LIN {X 0,Y 454.422,Z 912.402,A -85,B 0,C 180,E1 7856.185,E2 7856.185} C_VEL
LIN {X 0,Y 452.901,Z 864.791,A -85,B 0,C 180,E1 7857.267,E2 7857.267} C_VEL
LIN {X 0,Y 442.42,Z 831.81,A -85,B 0,C 180,E1 7858.557,E2 7858.557} C_VEL
LIN {X 0,Y 442.033,Z 831.81,A -85,B 0,C 180,E1 7869.429,E2 7869.429} C_VEL
LIN {X 0,Y 441.898,Z 831.81,A -85,B 0,C 180,E1 7877.954,E2 7877.954} C_VEL
LIN {X 0,Y 441.923,Z 831.81,A -85,B 0,C 180,E1 7887.837,E2 7887.837} C_VEL
LIN {X 0,Y 442.333,Z 831.81,A -85,B 0,C 180,E1 7898.882,E2 7898.882} C_VEL
LIN {X 0,Y 442.705,Z 831.81,A -85,B 0,C 180,E1 7909.13,E2 7909.13} C_VEL
LIN {X 0,Y 443.019,Z 831.81,A -85,B 0,C 180,E1 7919.017,E2 7919.017} C_VEL
LIN {X 0,Y 442.99,Z 831.81,A -85,B 0,C 180,E1 7928.866,E2 7928.866} C_VEL
LIN {X 0,Y 442.447,Z 831.81,A -85,B 0,C 180,E1 7939.4,E2 7939.4} C_VEL
LIN {X 0,Y 442.141,Z 831.81,A -85,B 0,C 180,E1 7949.846,E2 7949.846} C_VEL
LIN {X 0,Y 441.891,Z 831.81,A -85,B 0,C 180,E1 7959.444,E2 7959.444} C_VEL
LIN {X 0,Y 441.878,Z 831.81,A -85,B 0,C 180,E1 7967.957,E2 7967.957} C_VEL
LIN {X 0,Y 441.956,Z 831.81,A -85,B 0,C 180,E1 7977.844,E2 7977.844} C_VEL
LIN {X 0,Y 441.962,Z 831.81,A -85,B 0,C 180,E1 7986.742,E2 7986.742} C_VEL
LIN {X 0,Y 442.386,Z 831.81,A -85,B 0,C 180,E1 7997.116,E2 7997.116} C_VEL
LIN {X 0,Y 443.102,Z 831.81,A -85,B 0,C 180,E1 8007.055,E2 8007.055} C_VEL
LIN {X 0,Y 442.319,Z 833.399,A -85,B 0,C 180,E1 8012.396,E2 8012.396} C_VEL
LIN {X 0,Y 449.483,Z 869.862,A -85,B 0,C 180,E1 8014.631,E2 8014.631} C_VEL
LIN {X 0,Y 446.798,Z 905.325,A -85,B 0,C 180,E1 8018.299,E2 8018.299} C_VEL
LIN {X 0,Y 444.934,Z 929.395,A -85,B 0,C 180,E1 8023.352,E2 8023.352} C_VEL
LIN {X 0,Y 444.173,Z 939.173,A -85,B 0,C 180,E1 8028.939,E2 8028.939} C_VEL
LIN {X 0,Y 444.716,Z 934.706,A -85,B 0,C 180,E1 8034.709,E2 8034.709} C_VEL
LIN {X 0,Y 446.355,Z 916.606,A -85,B 0,C 180,E1 8039.89,E2 8039.89} C_VEL
LIN {X 0,Y 448.943,Z 886.147,A -85,B 0,C 180,E1 8044.088,E2 8044.088} C_VEL
LIN {X 0,Y 448.622,Z 854.294,A -85,B 0,C 180,E1 8046.544,E2 8046.544} C_VEL
LIN {X 0,Y 442.206,Z 831.81,A -85,B 0,C 180,E1 8047.897,E2 8047.897} C_VEL
LIN {X 0,Y 441.835,Z 831.81,A -85,B 0,C 180,E1 8057.952,E2 8057.952} C_VEL
LIN {X 0,Y 441.941,Z 831.81,A -85,B 0,C 180,E1 8067.843,E2 8067.843} C_VEL
LIN {X 0,Y 441.947,Z 831.81,A -85,B 0,C 180,E1 8076.742,E2 8076.742} C_VEL
LIN {X 0,Y 442.404,Z 831.81,A -85,B 0,C 180,E1 8087.118,E2 8087.118} C_VEL
LIN {X 0,Y 443.089,Z 831.81,A -85,B 0,C 180,E1 8097.057,E2 8097.057} C_VEL
LIN {X 0,Y 443.038,Z 831.81,A -85,B 0,C 180,E1 8106.888,E2 8106.888} C_VEL
LIN {X 0,Y 442.488,Z 831.81,A -85,B 0,C 180,E1 8116.952,E2 8116.952} C_VEL
LIN {X 0,Y 442.171,Z 831.81,A -85,B 0,C 180,E1 8127.606,E2 8127.606} C_VEL
LIN {X 0,Y 442.046,Z 831.81,A -85,B 0,C 180,E1 8136.93,E2 8136.93} C_VEL
LIN {X 0,Y 441.891,Z 831.81,A -85,B 0,C 180,E1 8147.598,E2 8147.598} C_VEL
LIN {X 0,Y 441.964,Z 831.81,A -85,B 0,C 180,E1 8157.845,E2 8157.845} C_VEL
LIN {X 0,Y 442.599,Z 833.755,A -85,B 0,C 180,E1 8161.637,E2 8161.637} C_VEL
LIN {X 0,Y 455.096,Z 877.398,A -85,B 0,C 180,E1 8163.05,E2 8163.05} C_VEL
LIN {X 0,Y 453.053,Z 934.016,A -85,B 0,C 180,E1 8164.683,E2 8164.683} C_VEL
LIN {X 0,Y 452.974,Z 934.968,A -85,B 0,C 180,E1 8164.729,E2 8164.729} C_VEL
LIN {X 0,Y 443.094,Z 966.571,A -85,B 0,C 180,E1 8166.367,E2 8166.367} C_VEL
LIN {X 0,Y 438.906,Z 1011.784,A -85,B 0,C 180,E1 8171.012,E2 8171.012} C_VEL
LIN {X 0,Y 436.535,Z 1045.486,A -85,B 0,C 180,E1 8176.941,E2 8176.941} C_VEL
LIN {X 0,Y 435.959,Z 1065.659,A -85,B 0,C 180,E1 8183.505,E2 8183.505} C_VEL
LIN {X 0,Y 436.168,Z 1071.941,A -85,B 0,C 180,E1 8189.004,E2 8189.004} C_VEL
LIN {X 0,Y 435.757,Z 1066.82,A -85,B 0,C 180,E1 8195.934,E2 8195.934} C_VEL
LIN {X 0,Y 436.23,Z 1047.781,A -85,B 0,C 180,E1 8202.558,E2 8202.558} C_VEL
LIN {X 0,Y 438.507,Z 1016.439,A -85,B 0,C 180,E1 8208.392,E2 8208.392} C_VEL
LIN {X 0,Y 442.634,Z 972.141,A -85,B 0,C 180,E1 8213.221,E2 8213.221} C_VEL
LIN {X 0,Y 446.471,Z 920.305,A -85,B 0,C 180,E1 8216.255,E2 8216.255} C_VEL
LIN {X 0,Y 445.695,Z 867.234,A -85,B 0,C 180,E1 8217.583,E2 8217.583} C_VEL
LIN {X 0,Y 434.365,Z 831.81,A -85,B 0,C 180,E1 8218.883,E2 8218.883} C_VEL
LIN {X 0,Y 433.936,Z 831.81,A -85,B 0,C 180,E1 8228.1,E2 8228.1} C_VEL
LIN {X 0,Y 433.837,Z 831.81,A -85,B 0,C 180,E1 8238.77,E2 8238.77} C_VEL
LIN {X 0,Y 433.955,Z 831.81,A -85,B 0,C 180,E1 8249.527,E2 8249.527} C_VEL
LIN {X 0,Y 434.401,Z 831.81,A -85,B 0,C 180,E1 8260.614,E2 8260.614} C_VEL
LIN {X 0,Y 434.81,Z 831.81,A -85,B 0,C 180,E1 8270.961,E2 8270.961} C_VEL
LIN {X 0,Y 435.516,Z 831.81,A -85,B 0,C 180,E1 8280.996,E2 8280.996} C_VEL
LIN {X 0,Y 434.775,Z 831.81,A -85,B 0,C 180,E1 8291.067,E2 8291.067} C_VEL
LIN {X 0,Y 434.374,Z 831.81,A -85,B 0,C 180,E1 8301.519,E2 8301.519} C_VEL
LIN {X 0,Y 433.976,Z 831.81,A -85,B 0,C 180,E1 8311.049,E2 8311.049} C_VEL
LIN {X 0,Y 433.808,Z 831.81,A -85,B 0,C 180,E1 8321.226,E2 8321.226} C_VEL
LIN {X 0,Y 433.755,Z 831.81,A -85,B 0,C 180,E1 8331.925,E2 8331.925} C_VEL
LIN {X 0,Y 434.054,Z 831.81,A -85,B 0,C 180,E1 8341.836,E2 8341.836} C_VEL
LIN {X 0,Y 434.263,Z 831.81,A -85,B 0,C 180,E1 8352.72,E2 8352.72} C_VEL
LIN {X 0,Y 434.922,Z 831.81,A -85,B 0,C 180,E1 8362.985,E2 8362.985} C_VEL
LIN {X 0,Y 434.261,Z 831.81,A -85,B 0,C 180,E1 8371.877,E2 8371.877} C_VEL
LIN {X 0,Y 441.916,Z 870.864,A -85,B 0,C 180,E1 8374.328,E2 8374.328} C_VEL
LIN {X 0,Y 439.148,Z 905.532,A -85,B 0,C 180,E1 8377.945,E2 8377.945} C_VEL
LIN {X 0,Y 437.129,Z 929.985,A -85,B 0,C 180,E1 8383.041,E2 8383.041} C_VEL
LIN {X 0,Y 436.474,Z 938.88,A -85,B 0,C 180,E1 8387.189,E2 8387.189} C_VEL
LIN {X 0,Y 436.668,Z 938.097,A -85,B 0,C 180,E1 8393.556,E2 8393.556} C_VEL
LIN {X 0,Y 438.194,Z 922.963,A -85,B 0,C 180,E1 8399.002,E2 8399.002} C_VEL
LIN {X 0,Y 440.773,Z 895,A -85,B 0,C 180,E1 8403.574,E2 8403.574} C_VEL
LIN {X 0,Y 441.368,Z 856.806,A -85,B 0,C 180,E1 8406.828,E2 8406.828} C_VEL
LIN {X 0,Y 434.167,Z 831.81,A -85,B 0,C 180,E1 8408.449,E2 8408.449} C_VEL
LIN {X 0,Y 433.703,Z 831.81,A -85,B 0,C 180,E1 8419.66,E2 8419.66} C_VEL
LIN {X 0,Y 433.965,Z 831.81,A -85,B 0,C 180,E1 8429.533,E2 8429.533} C_VEL
LIN {X 0,Y 434.066,Z 831.81,A -85,B 0,C 180,E1 8440.603,E2 8440.603} C_VEL
LIN {X 0,Y 434.843,Z 831.81,A -85,B 0,C 180,E1 8450.966,E2 8450.966} C_VEL
LIN {X 0,Y 435.008,Z 831.81,A -85,B 0,C 180,E1 8461.001,E2 8461.001} C_VEL
LIN {X 0,Y 434.712,Z 831.81,A -85,B 0,C 180,E1 8471.072,E2 8471.072} C_VEL
LIN {X 0,Y 434.335,Z 831.81,A -85,B 0,C 180,E1 8481.526,E2 8481.526} C_VEL
LIN {X 0,Y 433.993,Z 831.81,A -85,B 0,C 180,E1 8491.054,E2 8491.054} C_VEL
LIN {X 0,Y 433.899,Z 831.81,A -85,B 0,C 180,E1 8501.241,E2 8501.241} C_VEL
LIN {X 0,Y 433.843,Z 831.81,A -85,B 0,C 180,E1 8512.257,E2 8512.257} C_VEL
LIN {X 0,Y 434.468,Z 833.594,A -85,B 0,C 180,E1 8521.146,E2 8521.146} C_VEL
LIN {X 0,Y 447.732,Z 879.445,A -85,B 0,C 180,E1 8522.688,E2 8522.688} C_VEL
LIN {X 0,Y 445.41,Z 935.367,A -85,B 0,C 180,E1 8524.403,E2 8524.403} C_VEL
LIN {X 0,Y 443.094,Z 966.571,A -85,B 0,C 180,E1 8526.367,E2 8526.367} C_VEL
LIN {X 0,Y 432.74,Z 995.144,A -85,B 0,C 180,E1 8528.771,E2 8528.771} C_VEL
LIN {X 0,Y 429.368,Z 1034.587,A -85,B 0,C 180,E1 8534.629,E2 8534.629} C_VEL
LIN {X 0,Y 427.888,Z 1059.791,A -85,B 0,C 180,E1 8541.331,E2 8541.331} C_VEL
LIN {X 0,Y 427.788,Z 1069.446,A -85,B 0,C 180,E1 8546.95,E2 8546.95} C_VEL
LIN {X 0,Y 428.088,Z 1068.529,A -85,B 0,C 180,E1 8554.066,E2 8554.066} C_VEL
LIN {X 0,Y 428.186,Z 1052.254,A -85,B 0,C 180,E1 8561.241,E2 8561.241} C_VEL
LIN {X 0,Y 430.22,Z 1021.325,A -85,B 0,C 180,E1 8567.766,E2 8567.766} C_VEL
LIN {X 0,Y 434.404,Z 978.475,A -85,B 0,C 180,E1 8572.932,E2 8572.932} C_VEL
LIN {X 0,Y 438.433,Z 927.776,A -85,B 0,C 180,E1 8576.285,E2 8576.285} C_VEL
LIN {X 0,Y 438.872,Z 870.815,A -85,B 0,C 180,E1 8577.872,E2 8577.872} C_VEL
LIN {X 0,Y 426.276,Z 831.81,A -85,B 0,C 180,E1 8579.275,E2 8579.275} C_VEL
LIN {X 0,Y 425.881,Z 831.81,A -85,B 0,C 180,E1 8589.987,E2 8589.987} C_VEL
LIN {X 0,Y 425.797,Z 831.81,A -85,B 0,C 180,E1 8600.02,E2 8600.02} C_VEL
LIN {X 0,Y 425.943,Z 831.81,A -85,B 0,C 180,E1 8611.247,E2 8611.247} C_VEL
LIN {X 0,Y 426.421,Z 831.81,A -85,B 0,C 180,E1 8622.389,E2 8622.389} C_VEL
LIN {X 0,Y 426.997,Z 831.81,A -85,B 0,C 180,E1 8632.852,E2 8632.852} C_VEL
LIN {X 0,Y 427.059,Z 831.81,A -85,B 0,C 180,E1 8643.054,E2 8643.054} C_VEL
LIN {X 0,Y 426.64,Z 831.81,A -85,B 0,C 180,E1 8653.367,E2 8653.367} C_VEL
LIN {X 0,Y 426.262,Z 831.81,A -85,B 0,C 180,E1 8664.167,E2 8664.167} C_VEL
LIN {X 0,Y 425.868,Z 831.81,A -85,B 0,C 180,E1 8673.527,E2 8673.527} C_VEL
LIN {X 0,Y 425.807,Z 831.81,A -85,B 0,C 180,E1 8684.025,E2 8684.025} C_VEL
LIN {X 0,Y 425.75,Z 831.81,A -85,B 0,C 180,E1 8693.976,E2 8693.976} C_VEL
LIN {X 0,Y 426.032,Z 831.81,A -85,B 0,C 180,E1 8703.56,E2 8703.56} C_VEL
LIN {X 0,Y 426.321,Z 831.81,A -85,B 0,C 180,E1 8714.516,E2 8714.516} C_VEL
LIN {X 0,Y 426.823,Z 831.81,A -85,B 0,C 180,E1 8724.9,E2 8724.9} C_VEL
LIN {X 0,Y 426.5,Z 833.49,A -85,B 0,C 180,E1 8731.561,E2 8731.561} C_VEL
LIN {X 0,Y 434.317,Z 872.523,A -85,B 0,C 180,E1 8734.063,E2 8734.063} C_VEL
LIN {X 0,Y 431.356,Z 907.491,A -85,B 0,C 180,E1 8737.835,E2 8737.835} C_VEL
LIN {X 0,Y 429.326,Z 930.682,A -85,B 0,C 180,E1 8742.763,E2 8742.763} C_VEL
LIN {X 0,Y 428.543,Z 940.498,A -85,B 0,C 180,E1 8747.517,E2 8747.517} C_VEL
LIN {X 0,Y 428.749,Z 939.811,A -85,B 0,C 180,E1 8753.296,E2 8753.296} C_VEL
LIN {X 0,Y 430.281,Z 925.373,A -85,B 0,C 180,E1 8758.923,E2 8758.923} C_VEL
LIN {X 0,Y 432.969,Z 898.325,A -85,B 0,C 180,E1 8763.617,E2 8763.617} C_VEL
LIN {X 0,Y 434.419,Z 860.694,A -85,B 0,C 180,E1 8767.02,E2 8767.02} C_VEL
LIN {X 0,Y 426.096,Z 831.81,A -85,B 0,C 180,E1 8768.952,E2 8768.952} C_VEL
LIN {X 0,Y 425.672,Z 831.81,A -85,B 0,C 180,E1 8780.039,E2 8780.039} C_VEL
LIN {X 0,Y 425.956,Z 831.81,A -85,B 0,C 180,E1 8791.252,E2 8791.252} C_VEL
LIN {X 0,Y 426.191,Z 831.81,A -85,B 0,C 180,E1 8802.384,E2 8802.384} C_VEL
LIN {X 0,Y 426.9,Z 831.81,A -85,B 0,C 180,E1 8812.854,E2 8812.854} C_VEL
LIN {X 0,Y 427.017,Z 831.81,A -85,B 0,C 180,E1 8821.02,E2 8821.02} C_VEL
LIN {X 0,Y 426.69,Z 831.81,A -85,B 0,C 180,E1 8831.283,E2 8831.283} C_VEL
LIN {X 0,Y 426.3,Z 831.81,A -85,B 0,C 180,E1 8841.952,E2 8841.952} C_VEL
LIN {X 0,Y 425.973,Z 831.81,A -85,B 0,C 180,E1 8853.156,E2 8853.156} C_VEL
LIN {X 0,Y 425.852,Z 831.81,A -85,B 0,C 180,E1 8864.025,E2 8864.025} C_VEL
LIN {X 0,Y 425.799,Z 831.81,A -85,B 0,C 180,E1 8873.981,E2 8873.981} C_VEL
LIN {X 0,Y 426.336,Z 833.295,A -85,B 0,C 180,E1 8880.622,E2 8880.622} C_VEL
LIN {X 0,Y 440.369,Z 881.983,A -85,B 0,C 180,E1 8882.322,E2 8882.322} C_VEL
LIN {X 0,Y 437.735,Z 937.584,A -85,B 0,C 180,E1 8884.156,E2 8884.156} C_VEL
LIN {X 0,Y 433.497,Z 987.759,A -85,B 0,C 180,E1 8887.976,E2 8887.976} C_VEL
LIN {X 0,Y 432.74,Z 995.144,A -85,B 0,C 180,E1 8888.771,E2 8888.771} C_VEL
LIN {X 0,Y 422.54,Z 1019.728,A -85,B 0,C 180,E1 8891.909,E2 8891.909} C_VEL
LIN {X 0,Y 420.47,Z 1050.799,A -85,B 0,C 180,E1 8898.551,E2 8898.551} C_VEL
LIN {X 0,Y 419.97,Z 1067.213,A -85,B 0,C 180,E1 8905.856,E2 8905.856} C_VEL
LIN {X 0,Y 419.958,Z 1069.521,A -85,B 0,C 180,E1 8911.036,E2 8911.036} C_VEL
LIN {X 0,Y 419.861,Z 1061.159,A -85,B 0,C 180,E1 8917.79,E2 8917.79} C_VEL
LIN {X 0,Y 421.193,Z 1037.3,A -85,B 0,C 180,E1 8924.875,E2 8924.875} C_VEL
LIN {X 0,Y 424.412,Z 1000.57,A -85,B 0,C 180,E1 8930.814,E2 8930.814} C_VEL
LIN {X 0,Y 428.924,Z 952.896,A -85,B 0,C 180,E1 8935.219,E2 8935.219} C_VEL
LIN {X 0,Y 432.413,Z 900.477,A -85,B 0,C 180,E1 8937.613,E2 8937.613} C_VEL
LIN {X 0,Y 430.283,Z 868.597,A -85,B 0,C 180,E1 8938.364,E2 8938.364} C_VEL
LIN {X 0,Y 418.157,Z 831.81,A -85,B 0,C 180,E1 8939.936,E2 8939.936} C_VEL
LIN {X 0,Y 417.859,Z 831.81,A -85,B 0,C 180,E1 8949.461,E2 8949.461} C_VEL
LIN {X 0,Y 417.777,Z 831.81,A -85,B 0,C 180,E1 8960.525,E2 8960.525} C_VEL
LIN {X 0,Y 417.916,Z 831.81,A -85,B 0,C 180,E1 8970.641,E2 8970.641} C_VEL
LIN {X 0,Y 418.385,Z 831.81,A -85,B 0,C 180,E1 8982.04,E2 8982.04} C_VEL
LIN {X 0,Y 418.981,Z 831.81,A -85,B 0,C 180,E1 8992.715,E2 8992.715} C_VEL
LIN {X 0,Y 419.043,Z 831.81,A -85,B 0,C 180,E1 9003.112,E2 9003.112} C_VEL
LIN {X 0,Y 418.607,Z 831.81,A -85,B 0,C 180,E1 9013.628,E2 9013.628} C_VEL
LIN {X 0,Y 418.245,Z 831.81,A -85,B 0,C 180,E1 9024.661,E2 9024.661} C_VEL
LIN {X 0,Y 417.704,Z 831.81,A -85,B 0,C 180,E1 9035.17,E2 9035.17} C_VEL
LIN {X 0,Y 417.774,Z 831.81,A -85,B 0,C 180,E1 9045.099,E2 9045.099} C_VEL
LIN {X 0,Y 417.744,Z 831.81,A -85,B 0,C 180,E1 9055.731,E2 9055.731} C_VEL
LIN {X 0,Y 417.962,Z 831.81,A -85,B 0,C 180,E1 9065.32,E2 9065.32} C_VEL
LIN {X 0,Y 418.302,Z 831.81,A -85,B 0,C 180,E1 9076.36,E2 9076.36} C_VEL
LIN {X 0,Y 419.049,Z 831.81,A -85,B 0,C 180,E1 9086.886,E2 9086.886} C_VEL
LIN {X 0,Y 418.651,Z 833.62,A -85,B 0,C 180,E1 9091.135,E2 9091.135} C_VEL
LIN {X 0,Y 426.787,Z 873.187,A -85,B 0,C 180,E1 9093.713,E2 9093.713} C_VEL
LIN {X 0,Y 423.565,Z 909.392,A -85,B 0,C 180,E1 9097.721,E2 9097.721} C_VEL
LIN {X 0,Y 421.377,Z 932.957,A -85,B 0,C 180,E1 9103.006,E2 9103.006} C_VEL
LIN {X 0,Y 420.597,Z 942.014,A -85,B 0,C 180,E1 9107.859,E2 9107.859} C_VEL
LIN {X 0,Y 421.035,Z 939.377,A -85,B 0,C 180,E1 9114.487,E2 9114.487} C_VEL
LIN {X 0,Y 423.044,Z 922.373,A -85,B 0,C 180,E1 9120.126,E2 9120.126} C_VEL
LIN {X 0,Y 426.057,Z 893.863,A -85,B 0,C 180,E1 9124.61,E2 9124.61} C_VEL
LIN {X 0,Y 426.409,Z 859.686,A -85,B 0,C 180,E1 9127.602,E2 9127.602} C_VEL
LIN {X 0,Y 418.049,Z 831.81,A -85,B 0,C 180,E1 9129.439,E2 9129.439} C_VEL
LIN {X 0,Y 417.647,Z 831.81,A -85,B 0,C 180,E1 9140.515,E2 9140.515} C_VEL
LIN {X 0,Y 417.926,Z 831.81,A -85,B 0,C 180,E1 9150.647,E2 9150.647} C_VEL
LIN {X 0,Y 418.138,Z 831.81,A -85,B 0,C 180,E1 9162.033,E2 9162.033} C_VEL
LIN {X 0,Y 418.878,Z 831.81,A -85,B 0,C 180,E1 9172.717,E2 9172.717} C_VEL
LIN {X 0,Y 419.011,Z 831.81,A -85,B 0,C 180,E1 9181.04,E2 9181.04} C_VEL
LIN {X 0,Y 418.687,Z 831.81,A -85,B 0,C 180,E1 9191.502,E2 9191.502} C_VEL
LIN {X 0,Y 418.234,Z 831.81,A -85,B 0,C 180,E1 9202.398,E2 9202.398} C_VEL
LIN {X 0,Y 417.923,Z 831.81,A -85,B 0,C 180,E1 9211.775,E2 9211.775} C_VEL
LIN {X 0,Y 417.855,Z 831.81,A -85,B 0,C 180,E1 9222.218,E2 9222.218} C_VEL
LIN {X 0,Y 417.783,Z 831.81,A -85,B 0,C 180,E1 9233.178,E2 9233.178} C_VEL
LIN {X 0,Y 418.293,Z 833.427,A -85,B 0,C 180,E1 9240.09,E2 9240.09} C_VEL
LIN {X 0,Y 433.058,Z 882.531,A -85,B 0,C 180,E1 9241.906,E2 9241.906} C_VEL
LIN {X 0,Y 430.285,Z 936.811,A -85,B 0,C 180,E1 9243.747,E2 9243.747} C_VEL
LIN {X 0,Y 425.892,Z 986,A -85,B 0,C 180,E1 9247.534,E2 9247.534} C_VEL
LIN {X 0,Y 422.54,Z 1019.728,A -85,B 0,C 180,E1 9251.909,E2 9251.909} C_VEL
LIN {X 0,Y 412.802,Z 1039.684,A -85,B 0,C 180,E1 9255.728,E2 9255.728} C_VEL
LIN {X 0,Y 412.014,Z 1060.915,A -85,B 0,C 180,E1 9262.594,E2 9262.594} C_VEL
LIN {X 0,Y 412.387,Z 1068.355,A -85,B 0,C 180,E1 9268.946,E2 9268.946} C_VEL
LIN {X 0,Y 411.912,Z 1063.046,A -85,B 0,C 180,E1 9276.351,E2 9276.351} C_VEL
LIN {X 0,Y 412.463,Z 1044.474,A -85,B 0,C 180,E1 9283.123,E2 9283.123} C_VEL
LIN {X 0,Y 414.97,Z 1013.498,A -85,B 0,C 180,E1 9289.216,E2 9289.216} C_VEL
LIN {X 0,Y 419.687,Z 969.196,A -85,B 0,C 180,E1 9294.287,E2 9294.287} C_VEL
LIN {X 0,Y 424.093,Z 917.458,A -85,B 0,C 180,E1 9297.432,E2 9297.432} C_VEL
LIN {X 0,Y 423.379,Z 871.81,A -85,B 0,C 180,E1 9298.683,E2 9298.683} C_VEL
LIN {X 0,Y 410.125,Z 831.81,A -85,B 0,C 180,E1 9300.234,E2 9300.234} C_VEL
LIN {X 0,Y 409.773,Z 831.81,A -85,B 0,C 180,E1 9310.6,E2 9310.6} C_VEL
LIN {X 0,Y 409.709,Z 831.81,A -85,B 0,C 180,E1 9319.589,E2 9319.589} C_VEL
LIN {X 0,Y 409.896,Z 831.81,A -85,B 0,C 180,E1 9330.463,E2 9330.463} C_VEL
LIN {X 0,Y 410.325,Z 831.81,A -85,B 0,C 180,E1 9341.674,E2 9341.674} C_VEL
LIN {X 0,Y 410.944,Z 831.81,A -85,B 0,C 180,E1 9352.571,E2 9352.571} C_VEL
LIN {X 0,Y 411.04,Z 831.81,A -85,B 0,C 180,E1 9363.173,E2 9363.173} C_VEL
LIN {X 0,Y 410.57,Z 831.81,A -85,B 0,C 180,E1 9373.9,E2 9373.9} C_VEL
LIN {X 0,Y 410.153,Z 831.81,A -85,B 0,C 180,E1 9385.181,E2 9385.181} C_VEL
LIN {X 0,Y 409.708,Z 831.81,A -85,B 0,C 180,E1 9395.037,E2 9395.037} C_VEL
LIN {X 0,Y 409.67,Z 831.81,A -85,B 0,C 180,E1 9406.248,E2 9406.248} C_VEL
LIN {X 0,Y 409.747,Z 831.81,A -85,B 0,C 180,E1 9417.518,E2 9417.518} C_VEL
LIN {X 0,Y 409.854,Z 831.81,A -85,B 0,C 180,E1 9427.121,E2 9427.121} C_VEL
LIN {X 0,Y 410.464,Z 831.81,A -85,B 0,C 180,E1 9438.454,E2 9438.454} C_VEL
LIN {X 0,Y 411.311,Z 831.81,A -85,B 0,C 180,E1 9448.943,E2 9448.943} C_VEL
LIN {X 0,Y 410.796,Z 833.812,A -85,B 0,C 180,E1 9450.694,E2 9450.694} C_VEL
LIN {X 0,Y 419.233,Z 874.42,A -85,B 0,C 180,E1 9453.402,E2 9453.402} C_VEL
LIN {X 0,Y 415.938,Z 909.617,A -85,B 0,C 180,E1 9457.336,E2 9457.336} C_VEL
LIN {X 0,Y 413.628,Z 933.1,A -85,B 0,C 180,E1 9462.526,E2 9462.526} C_VEL
LIN {X 0,Y 412.652,Z 943.528,A -85,B 0,C 180,E1 9468.215,E2 9468.215} C_VEL
LIN {X 0,Y 413.255,Z 939.955,A -85,B 0,C 180,E1 9474.979,E2 9474.979} C_VEL
LIN {X 0,Y 415.541,Z 921.312,A -85,B 0,C 180,E1 9480.882,E2 9480.882} C_VEL
LIN {X 0,Y 419.021,Z 890.846,A -85,B 0,C 180,E1 9485.425,E2 9485.425} C_VEL
LIN {X 0,Y 418.779,Z 860.336,A -85,B 0,C 180,E1 9488.073,E2 9488.073} C_VEL
LIN {X 0,Y 409.908,Z 831.81,A -85,B 0,C 180,E1 9490.167,E2 9490.167} C_VEL
LIN {X 0,Y 409.605,Z 831.81,A -85,B 0,C 180,E1 9499.582,E2 9499.582} C_VEL
LIN {X 0,Y 409.917,Z 831.81,A -85,B 0,C 180,E1 9510.456,E2 9510.456} C_VEL
LIN {X 0,Y 410.06,Z 831.81,A -85,B 0,C 180,E1 9521.666,E2 9521.666} C_VEL
LIN {X 0,Y 410.849,Z 831.81,A -85,B 0,C 180,E1 9532.574,E2 9532.574} C_VEL
LIN {X 0,Y 411.02,Z 831.81,A -85,B 0,C 180,E1 9541.06,E2 9541.06} C_VEL
LIN {X 0,Y 410.679,Z 831.81,A -85,B 0,C 180,E1 9551.729,E2 9551.729} C_VEL
LIN {X 0,Y 410.169,Z 831.81,A -85,B 0,C 180,E1 9562.864,E2 9562.864} C_VEL
LIN {X 0,Y 409.818,Z 831.81,A -85,B 0,C 180,E1 9573.575,E2 9573.575} C_VEL
LIN {X 0,Y 409.714,Z 831.81,A -85,B 0,C 180,E1 9583.759,E2 9583.759} C_VEL
LIN {X 0,Y 409.737,Z 831.81,A -85,B 0,C 180,E1 9594.966,E2 9594.966} C_VEL
LIN {X 0,Y 410.286,Z 833.663,A -85,B 0,C 180,E1 9599.527,E2 9599.527} C_VEL
LIN {X 0,Y 425.783,Z 883.698,A -85,B 0,C 180,E1 9601.48,E2 9601.48} C_VEL
LIN {X 0,Y 422.731,Z 937.734,A -85,B 0,C 180,E1 9603.41,E2 9603.41} C_VEL
LIN {X 0,Y 417.973,Z 987.695,A -85,B 0,C 180,E1 9607.45,E2 9607.45} C_VEL
LIN {X 0,Y 414.091,Z 1028.005,A -85,B 0,C 180,E1 9613.26,E2 9613.26} C_VEL
LIN {X 0,Y 412.802,Z 1039.684,A -85,B 0,C 180,E1 9615.728,E2 9615.728} C_VEL
LIN {X 0,Y 404.265,Z 1054.28,A -85,B 0,C 180,E1 9620.126,E2 9620.126} C_VEL
LIN {X 0,Y 404.059,Z 1065.854,A -85,B 0,C 180,E1 9626.771,E2 9626.771} C_VEL
LIN {X 0,Y 404.291,Z 1064.897,A -85,B 0,C 180,E1 9634.306,E2 9634.306} C_VEL
LIN {X 0,Y 404.267,Z 1050.07,A -85,B 0,C 180,E1 9641.366,E2 9641.366} C_VEL
LIN {X 0,Y 406.332,Z 1021.45,A -85,B 0,C 180,E1 9648.022,E2 9648.022} C_VEL
LIN {X 0,Y 410.897,Z 980.22,A -85,B 0,C 180,E1 9653.537,E2 9653.537} C_VEL
LIN {X 0,Y 415.595,Z 930.179,A -85,B 0,C 180,E1 9657.231,E2 9657.231} C_VEL
LIN {X 0,Y 416.669,Z 875.936,A -85,B 0,C 180,E1 9658.978,E2 9658.978} C_VEL
LIN {X 0,Y 402.095,Z 831.81,A -85,B 0,C 180,E1 9660.631,E2 9660.631} C_VEL
LIN {X 0,Y 401.674,Z 831.81,A -85,B 0,C 180,E1 9671.389,E2 9671.389} C_VEL
LIN {X 0,Y 401.642,Z 831.81,A -85,B 0,C 180,E1 9681.428,E2 9681.428} C_VEL
LIN {X 0,Y 401.909,Z 831.81,A -85,B 0,C 180,E1 9692.539,E2 9692.539} C_VEL
LIN {X 0,Y 402.484,Z 831.81,A -85,B 0,C 180,E1 9704.043,E2 9704.043} C_VEL
LIN {X 0,Y 402.993,Z 831.81,A -85,B 0,C 180,E1 9714.596,E2 9714.596} C_VEL
LIN {X 0,Y 402.951,Z 831.81,A -85,B 0,C 180,E1 9723.613,E2 9723.613} C_VEL
LIN {X 0,Y 402.535,Z 831.81,A -85,B 0,C 180,E1 9734.183,E2 9734.183} C_VEL
LIN {X 0,Y 402.066,Z 831.81,A -85,B 0,C 180,E1 9745.724,E2 9745.724} C_VEL
LIN {X 0,Y 401.646,Z 831.81,A -85,B 0,C 180,E1 9755.848,E2 9755.848} C_VEL
LIN {X 0,Y 401.608,Z 831.81,A -85,B 0,C 180,E1 9765.649,E2 9765.649} C_VEL
LIN {X 0,Y 401.711,Z 831.81,A -85,B 0,C 180,E1 9776.786,E2 9776.786} C_VEL
LIN {X 0,Y 401.837,Z 831.81,A -85,B 0,C 180,E1 9787.708,E2 9787.708} C_VEL
LIN {X 0,Y 402.392,Z 831.81,A -85,B 0,C 180,E1 9798.028,E2 9798.028} C_VEL
LIN {X 0,Y 403.301,Z 831.81,A -85,B 0,C 180,E1 9808.922,E2 9808.922} C_VEL
LIN {X 0,Y 403.002,Z 833.939,A -85,B 0,C 180,E1 9810.236,E2 9810.236} C_VEL
LIN {X 0,Y 411.716,Z 875.082,A -85,B 0,C 180,E1 9813.038,E2 9813.038} C_VEL
LIN {X 0,Y 408.14,Z 911.447,A -85,B 0,C 180,E1 9817.209,E2 9817.209} C_VEL
LIN {X 0,Y 405.721,Z 935.024,A -85,B 0,C 180,E1 9822.664,E2 9822.664} C_VEL
LIN {X 0,Y 404.734,Z 944.938,A -85,B 0,C 180,E1 9828.584,E2 9828.584} C_VEL
LIN {X 0,Y 405.447,Z 940.499,A -85,B 0,C 180,E1 9835.494,E2 9835.494} C_VEL
LIN {X 0,Y 407.953,Z 921.631,A -85,B 0,C 180,E1 9841.344,E2 9841.344} C_VEL
LIN {X 0,Y 411.719,Z 890.66,A -85,B 0,C 180,E1 9845.945,E2 9845.945} C_VEL
LIN {X 0,Y 411.583,Z 862.876,A -85,B 0,C 180,E1 9848.416,E2 9848.416} C_VEL
LIN {X 0,Y 401.812,Z 831.81,A -85,B 0,C 180,E1 9850.931,E2 9850.931} C_VEL
LIN {X 0,Y 401.499,Z 831.81,A -85,B 0,C 180,E1 9861.417,E2 9861.417} C_VEL
LIN {X 0,Y 401.911,Z 831.81,A -85,B 0,C 180,E1 9872.537,E2 9872.537} C_VEL
LIN {X 0,Y 402.229,Z 831.81,A -85,B 0,C 180,E1 9884.167,E2 9884.167} C_VEL
LIN {X 0,Y 402.806,Z 831.81,A -85,B 0,C 180,E1 9894.597,E2 9894.597} C_VEL
LIN {X 0,Y 402.879,Z 831.81,A -85,B 0,C 180,E1 9903.46,E2 9903.46} C_VEL
LIN {X 0,Y 402.543,Z 831.81,A -85,B 0,C 180,E1 9914.187,E2 9914.187} C_VEL
LIN {X 0,Y 402.023,Z 831.81,A -85,B 0,C 180,E1 9925.732,E2 9925.732} C_VEL
LIN {X 0,Y 401.798,Z 831.81,A -85,B 0,C 180,E1 9935.837,E2 9935.837} C_VEL
LIN {X 0,Y 401.638,Z 831.81,A -85,B 0,C 180,E1 9945.654,E2 9945.654} C_VEL
LIN {X 0,Y 401.736,Z 831.81,A -85,B 0,C 180,E1 9956.789,E2 9956.789} C_VEL
LIN {X 0,Y 402.193,Z 833.57,A -85,B 0,C 180,E1 9958.92,E2 9958.92} C_VEL
LIN {X 0,Y 418.532,Z 883.85,A -85,B 0,C 180,E1 9961.021,E2 9961.021} C_VEL
LIN {X 0,Y 415.326,Z 937.504,A -85,B 0,C 180,E1 9962.994,E2 9962.994} C_VEL
LIN {X 0,Y 410.358,Z 986.281,A -85,B 0,C 180,E1 9967.008,E2 9967.008} C_VEL
LIN {X 0,Y 406.217,Z 1026.846,A -85,B 0,C 180,E1 9972.955,E2 9972.955} C_VEL
LIN {X 0,Y 404.265,Z 1054.28,A -85,B 0,C 180,E1 9980.126,E2 9980.126} C_VEL
LIN {X 0,Y 396.284,Z 1062.81,A -85,B 0,C 180,E1 9984.942,E2 9984.942} C_VEL
LIN {X 0,Y 396.225,Z 1065.94,A -85,B 0,C 180,E1 9991.098,E2 9991.098} C_VEL
LIN {X 0,Y 396.115,Z 1057.386,A -85,B 0,C 180,E1 9998.26,E2 9998.26} C_VEL
LIN {X 0,Y 397.702,Z 1033.036,A -85,B 0,C 180,E1 10005.776,E2 10005.776} C_VEL
LIN {X 0,Y 401.455,Z 995.539,A -85,B 0,C 180,E1 10012.04,E2 10012.04} C_VEL
LIN {X 0,Y 406.55,Z 947.581,A -85,B 0,C 180,E1 10016.557,E2 10016.557} C_VEL
LIN {X 0,Y 410.233,Z 895.116,A -85,B 0,C 180,E1 10018.932,E2 10018.932} C_VEL
LIN {X 0,Y 407.173,Z 870.658,A -85,B 0,C 180,E1 10019.612,E2 10019.612} C_VEL
LIN {X 0,Y 393.963,Z 831.81,A -85,B 0,C 180,E1 10021.334,E2 10021.334} C_VEL
LIN {X 0,Y 393.659,Z 831.81,A -85,B 0,C 180,E1 10032.425,E2 10032.425} C_VEL
LIN {X 0,Y 393.567,Z 831.81,A -85,B 0,C 180,E1 10043.292,E2 10043.292} C_VEL
LIN {X 0,Y 393.871,Z 831.81,A -85,B 0,C 180,E1 10053.695,E2 10053.695} C_VEL
LIN {X 0,Y 394.539,Z 831.81,A -85,B 0,C 180,E1 10065.519,E2 10065.519} C_VEL
LIN {X 0,Y 394.919,Z 831.81,A -85,B 0,C 180,E1 10076.693,E2 10076.693} C_VEL
LIN {X 0,Y 394.814,Z 831.81,A -85,B 0,C 180,E1 10085.512,E2 10085.512} C_VEL
LIN {X 0,Y 394.46,Z 831.81,A -85,B 0,C 180,E1 10096.769,E2 10096.769} C_VEL
LIN {X 0,Y 394.028,Z 831.81,A -85,B 0,C 180,E1 10106.289,E2 10106.289} C_VEL
LIN {X 0,Y 393.522,Z 831.81,A -85,B 0,C 180,E1 10117.763,E2 10117.763} C_VEL
LIN {X 0,Y 393.554,Z 831.81,A -85,B 0,C 180,E1 10128.757,E2 10128.757} C_VEL
LIN {X 0,Y 393.721,Z 831.81,A -85,B 0,C 180,E1 10140.14,E2 10140.14} C_VEL
LIN {X 0,Y 393.939,Z 831.81,A -85,B 0,C 180,E1 10150.886,E2 10150.886} C_VEL
LIN {X 0,Y 394.783,Z 831.81,A -85,B 0,C 180,E1 10162.268,E2 10162.268} C_VEL
LIN {X 0,Y 395.022,Z 833.052,A -85,B 0,C 180,E1 10169.724,E2 10169.724} C_VEL
LIN {X 0,Y 404.224,Z 875.741,A -85,B 0,C 180,E1 10172.661,E2 10172.661} C_VEL
LIN {X 0,Y 400.58,Z 911.608,A -85,B 0,C 180,E1 10176.799,E2 10176.799} C_VEL
LIN {X 0,Y 398.016,Z 934.968,A -85,B 0,C 180,E1 10182.104,E2 10182.104} C_VEL
LIN {X 0,Y 397.081,Z 944.396,A -85,B 0,C 180,E1 10186.656,E2 10186.656} C_VEL
LIN {X 0,Y 396.863,Z 946.437,A -85,B 0,C 180,E1 10191.3,E2 10191.3} C_VEL
LIN {X 0,Y 398.222,Z 936.677,A -85,B 0,C 180,E1 10197.852,E2 10197.852} C_VEL
LIN {X 0,Y 401.482,Z 913.185,A -85,B 0,C 180,E1 10203.477,E2 10203.477} C_VEL
LIN {X 0,Y 405.58,Z 877.859,A -85,B 0,C 180,E1 10207.687,E2 10207.687} C_VEL
LIN {X 0,Y 397.574,Z 842.646,A -85,B 0,C 180,E1 10210.568,E2 10210.568} C_VEL
LIN {X 0,Y 393.762,Z 831.81,A -85,B 0,C 180,E1 10211.277,E2 10211.277} C_VEL
LIN {X 0,Y 393.432,Z 831.81,A -85,B 0,C 180,E1 10222.252,E2 10222.252} C_VEL
LIN {X 0,Y 393.852,Z 831.81,A -85,B 0,C 180,E1 10233.699,E2 10233.699} C_VEL
LIN {X 0,Y 394.23,Z 831.81,A -85,B 0,C 180,E1 10245.511,E2 10245.511} C_VEL
LIN {X 0,Y 395.024,Z 831.81,A -85,B 0,C 180,E1 10256.699,E2 10256.699} C_VEL
LIN {X 0,Y 394.883,Z 831.81,A -85,B 0,C 180,E1 10267.733,E2 10267.733} C_VEL
LIN {X 0,Y 394.248,Z 831.81,A -85,B 0,C 180,E1 10279.101,E2 10279.101} C_VEL
LIN {X 0,Y 393.802,Z 831.81,A -85,B 0,C 180,E1 10289.883,E2 10289.883} C_VEL
LIN {X 0,Y 393.652,Z 831.81,A -85,B 0,C 180,E1 10301.26,E2 10301.26} C_VEL
LIN {X 0,Y 393.558,Z 831.81,A -85,B 0,C 180,E1 10312.237,E2 10312.237} C_VEL
LIN {X 0,Y 394.058,Z 833.428,A -85,B 0,C 180,E1 10318.279,E2 10318.279} C_VEL
LIN {X 0,Y 411.329,Z 883.93,A -85,B 0,C 180,E1 10320.544,E2 10320.544} C_VEL
LIN {X 0,Y 407.89,Z 937.583,A -85,B 0,C 180,E1 10322.58,E2 10322.58} C_VEL
LIN {X 0,Y 402.647,Z 986.127,A -85,B 0,C 180,E1 10326.689,E2 10326.689} C_VEL
LIN {X 0,Y 398.318,Z 1025.921,A -85,B 0,C 180,E1 10332.684,E2 10332.684} C_VEL
LIN {X 0,Y 396.316,Z 1053.59,A -85,B 0,C 180,E1 10340.129,E2 10340.129} C_VEL
LIN {X 0,Y 396.284,Z 1062.81,A -85,B 0,C 180,E1 10344.942,E2 10344.942} C_VEL
LIN {X 0,Y 388.381,Z 1064.754,A -85,B 0,C 180,E1 10349.988,E2 10349.988} C_VEL
LIN {X 0,Y 388.098,Z 1058.297,A -85,B 0,C 180,E1 10357.301,E2 10357.301} C_VEL
LIN {X 0,Y 389.063,Z 1037.513,A -85,B 0,C 180,E1 10364.687,E2 10364.687} C_VEL
LIN {X 0,Y 392.74,Z 1001.917,A -85,B 0,C 180,E1 10371.387,E2 10371.387} C_VEL
LIN {X 0,Y 397.95,Z 956.706,A -85,B 0,C 180,E1 10376.232,E2 10376.232} C_VEL
LIN {X 0,Y 402.455,Z 904.005,A -85,B 0,C 180,E1 10379.086,E2 10379.086} C_VEL
LIN {X 0,Y 400.759,Z 875.43,A -85,B 0,C 180,E1 10379.907,E2 10379.907} C_VEL
LIN {X 0,Y 385.881,Z 831.81,A -85,B 0,C 180,E1 10381.739,E2 10381.739} C_VEL
LIN {X 0,Y 385.627,Z 831.81,A -85,B 0,C 180,E1 10393.525,E2 10393.525} C_VEL
LIN {X 0,Y 385.547,Z 831.81,A -85,B 0,C 180,E1 10405.194,E2 10405.194} C_VEL
LIN {X 0,Y 385.897,Z 831.81,A -85,B 0,C 180,E1 10415.608,E2 10415.608} C_VEL
LIN {X 0,Y 386.476,Z 831.81,A -85,B 0,C 180,E1 10425.21,E2 10425.21} C_VEL
LIN {X 0,Y 386.932,Z 831.81,A -85,B 0,C 180,E1 10436.625,E2 10436.625} C_VEL
LIN {X 0,Y 386.833,Z 831.81,A -85,B 0,C 180,E1 10445.626,E2 10445.626} C_VEL
LIN {X 0,Y 386.399,Z 831.81,A -85,B 0,C 180,E1 10457.13,E2 10457.13} C_VEL
LIN {X 0,Y 385.872,Z 831.81,A -85,B 0,C 180,E1 10467.764,E2 10467.764} C_VEL
LIN {X 0,Y 385.535,Z 831.81,A -85,B 0,C 180,E1 10479.864,E2 10479.864} C_VEL
LIN {X 0,Y 385.507,Z 831.81,A -85,B 0,C 180,E1 10490.141,E2 10490.141} C_VEL
LIN {X 0,Y 385.726,Z 831.81,A -85,B 0,C 180,E1 10500.542,E2 10500.542} C_VEL
LIN {X 0,Y 385.894,Z 831.81,A -85,B 0,C 180,E1 10510.472,E2 10510.472} C_VEL
LIN {X 0,Y 386.747,Z 831.81,A -85,B 0,C 180,E1 10522.106,E2 10522.106} C_VEL
LIN {X 0,Y 387.325,Z 833.718,A -85,B 0,C 180,E1 10529.262,E2 10529.262} C_VEL
LIN {X 0,Y 396.767,Z 875.85,A -85,B 0,C 180,E1 10532.225,E2 10532.225} C_VEL
LIN {X 0,Y 393.005,Z 911.728,A -85,B 0,C 180,E1 10536.373,E2 10536.373} C_VEL
LIN {X 0,Y 390.236,Z 935.579,A -85,B 0,C 180,E1 10541.78,E2 10541.78} C_VEL
LIN {X 0,Y 389.084,Z 946.177,A -85,B 0,C 180,E1 10547.14,E2 10547.14} C_VEL
LIN {X 0,Y 389.451,Z 945.448,A -85,B 0,C 180,E1 10554.151,E2 10554.151} C_VEL
LIN {X 0,Y 391.971,Z 929.851,A -85,B 0,C 180,E1 10560.542,E2 10560.542} C_VEL
LIN {X 0,Y 395.986,Z 901.243,A -85,B 0,C 180,E1 10565.772,E2 10565.772} C_VEL
LIN {X 0,Y 397.245,Z 867.797,A -85,B 0,C 180,E1 10569.154,E2 10569.154} C_VEL
LIN {X 0,Y 385.658,Z 831.81,A -85,B 0,C 180,E1 10572.208,E2 10572.208} C_VEL
LIN {X 0,Y 385.433,Z 831.81,A -85,B 0,C 180,E1 10583.816,E2 10583.816} C_VEL
LIN {X 0,Y 385.761,Z 831.81,A -85,B 0,C 180,E1 10593.103,E2 10593.103} C_VEL
LIN {X 0,Y 386.177,Z 831.81,A -85,B 0,C 180,E1 10605.203,E2 10605.203} C_VEL
LIN {X 0,Y 387.022,Z 831.81,A -85,B 0,C 180,E1 10616.63,E2 10616.63} C_VEL
LIN {X 0,Y 386.846,Z 831.81,A -85,B 0,C 180,E1 10627.894,E2 10627.894} C_VEL
LIN {X 0,Y 386.219,Z 831.81,A -85,B 0,C 180,E1 10639.514,E2 10639.514} C_VEL
LIN {X 0,Y 385.84,Z 831.81,A -85,B 0,C 180,E1 10649.453,E2 10649.453} C_VEL
LIN {X 0,Y 385.612,Z 831.81,A -85,B 0,C 180,E1 10660.498,E2 10660.498} C_VEL
LIN {X 0,Y 385.565,Z 831.81,A -85,B 0,C 180,E1 10670.137,E2 10670.137} C_VEL
LIN {X 0,Y 385.978,Z 833.558,A -85,B 0,C 180,E1 10677.601,E2 10677.601} C_VEL
LIN {X 0,Y 404.188,Z 885.852,A -85,B 0,C 180,E1 10680.079,E2 10680.079} C_VEL
LIN {X 0,Y 400.342,Z 939.314,A -85,B 0,C 180,E1 10682.249,E2 10682.249} C_VEL
LIN {X 0,Y 394.789,Z 987.262,A -85,B 0,C 180,E1 10686.508,E2 10686.508} C_VEL
LIN {X 0,Y 390.34,Z 1026.164,A -85,B 0,C 180,E1 10692.627,E2 10692.627} C_VEL
LIN {X 0,Y 388.394,Z 1052.241,A -85,B 0,C 180,E1 10699.874,E2 10699.874} C_VEL
LIN {X 0,Y 388.242,Z 1063.479,A -85,B 0,C 180,E1 10706.639,E2 10706.639} C_VEL
LIN {X 0,Y 388.381,Z 1064.754,A -85,B 0,C 180,E1 10709.988,E2 10709.988} C_VEL
LIN {X 0,Y 380.356,Z 1060.541,A -85,B 0,C 180,E1 10715.123,E2 10715.123} C_VEL
LIN {X 0,Y 380.445,Z 1044.196,A -85,B 0,C 180,E1 10722.673,E2 10722.673} C_VEL
LIN {X 0,Y 383.177,Z 1013.855,A -85,B 0,C 180,E1 10729.672,E2 10729.672} C_VEL
LIN {X 0,Y 388.595,Z 971.141,A -85,B 0,C 180,E1 10735.286,E2 10735.286} C_VEL
LIN {X 0,Y 393.846,Z 920.558,A -85,B 0,C 180,E1 10738.849,E2 10738.849} C_VEL
LIN {X 0,Y 393.753,Z 878.281,A -85,B 0,C 180,E1 10740.273,E2 10740.273} C_VEL
LIN {X 0,Y 377.823,Z 831.81,A -85,B 0,C 180,E1 10742.304,E2 10742.304} C_VEL
LIN {X 0,Y 377.512,Z 831.81,A -85,B 0,C 180,E1 10751.948,E2 10751.948} C_VEL
LIN {X 0,Y 377.498,Z 831.81,A -85,B 0,C 180,E1 10761.62,E2 10761.62} C_VEL
LIN {X 0,Y 377.744,Z 831.81,A -85,B 0,C 180,E1 10772.479,E2 10772.479} C_VEL
LIN {X 0,Y 378.242,Z 831.81,A -85,B 0,C 180,E1 10782.484,E2 10782.484} C_VEL
LIN {X 0,Y 378.943,Z 831.81,A -85,B 0,C 180,E1 10794.251,E2 10794.251} C_VEL
LIN {X 0,Y 379.009,Z 831.81,A -85,B 0,C 180,E1 10803.441,E2 10803.441} C_VEL
LIN {X 0,Y 378.464,Z 831.81,A -85,B 0,C 180,E1 10815.106,E2 10815.106} C_VEL
LIN {X 0,Y 377.939,Z 831.81,A -85,B 0,C 180,E1 10825.385,E2 10825.385} C_VEL
LIN {X 0,Y 377.489,Z 831.81,A -85,B 0,C 180,E1 10835.655,E2 10835.655} C_VEL
LIN {X 0,Y 377.418,Z 831.81,A -85,B 0,C 180,E1 10845.279,E2 10845.279} C_VEL
LIN {X 0,Y 377.552,Z 831.81,A -85,B 0,C 180,E1 10857.137,E2 10857.137} C_VEL
LIN {X 0,Y 377.773,Z 831.81,A -85,B 0,C 180,E1 10867.565,E2 10867.565} C_VEL
LIN {X 0,Y 378.516,Z 831.81,A -85,B 0,C 180,E1 10879.606,E2 10879.606} C_VEL
LIN {X 0,Y 379.407,Z 833.177,A -85,B 0,C 180,E1 10888.725,E2 10888.725} C_VEL
LIN {X 0,Y 389.262,Z 876.439,A -85,B 0,C 180,E1 10891.821,E2 10891.821} C_VEL
LIN {X 0,Y 385.443,Z 911.772,A -85,B 0,C 180,E1 10895.932,E2 10895.932} C_VEL
LIN {X 0,Y 382.443,Z 936.164,A -85,B 0,C 180,E1 10901.443,E2 10901.443} C_VEL
LIN {X 0,Y 381.15,Z 947.623,A -85,B 0,C 180,E1 10907.374,E2 10907.374} C_VEL
LIN {X 0,Y 381.365,Z 947.891,A -85,B 0,C 180,E1 10913.112,E2 10913.112} C_VEL
LIN {X 0,Y 383.555,Z 935.205,A -85,B 0,C 180,E1 10919.641,E2 10919.641} C_VEL
LIN {X 0,Y 387.593,Z 909.112,A -85,B 0,C 180,E1 10925.232,E2 10925.232} C_VEL
LIN {X 0,Y 390.614,Z 872.825,A -85,B 0,C 180,E1 10929.287,E2 10929.287} C_VEL
LIN {X 0,Y 377.602,Z 831.81,A -85,B 0,C 180,E1 10932.769,E2 10932.769} C_VEL
LIN {X 0,Y 377.427,Z 831.81,A -85,B 0,C 180,E1 10944.338,E2 10944.338} C_VEL
LIN {X 0,Y 377.727,Z 831.81,A -85,B 0,C 180,E1 10955.05,E2 10955.05} C_VEL
LIN {X 0,Y 378.156,Z 831.81,A -85,B 0,C 180,E1 10964.881,E2 10964.881} C_VEL
LIN {X 0,Y 379.001,Z 831.81,A -85,B 0,C 180,E1 10976.559,E2 10976.559} C_VEL
LIN {X 0,Y 378.81,Z 831.81,A -85,B 0,C 180,E1 10988.063,E2 10988.063} C_VEL
LIN {X 0,Y 378.148,Z 831.81,A -85,B 0,C 180,E1 10999.948,E2 10999.948} C_VEL
LIN {X 0,Y 377.723,Z 831.81,A -85,B 0,C 180,E1 11010.257,E2 11010.257} C_VEL
LIN {X 0,Y 377.505,Z 831.81,A -85,B 0,C 180,E1 11021.954,E2 11021.954} C_VEL
LIN {X 0,Y 377.497,Z 831.81,A -85,B 0,C 180,E1 11031.627,E2 11031.627} C_VEL
LIN {X 0,Y 377.983,Z 833.733,A -85,B 0,C 180,E1 11036.895,E2 11036.895} C_VEL
LIN {X 0,Y 397.06,Z 886.732,A -85,B 0,C 180,E1 11039.573,E2 11039.573} C_VEL
LIN {X 0,Y 392.912,Z 940.146,A -85,B 0,C 180,E1 11041.841,E2 11041.841} C_VEL
LIN {X 0,Y 387.008,Z 987.898,A -85,B 0,C 180,E1 11046.258,E2 11046.258} C_VEL
LIN {X 0,Y 382.321,Z 1026.938,A -85,B 0,C 180,E1 11052.681,E2 11052.681} C_VEL
LIN {X 0,Y 380.382,Z 1052.477,A -85,B 0,C 180,E1 11060.239,E2 11060.239} C_VEL
LIN {X 0,Y 380.32,Z 1062.288,A -85,B 0,C 180,E1 11066.569,E2 11066.569} C_VEL
LIN {X 0,Y 380.426,Z 1062.278,A -85,B 0,C 180,E1 11073.431,E2 11073.431} C_VEL
LIN {X 0,Y 380.356,Z 1060.541,A -85,B 0,C 180,E1 11075.123,E2 11075.123} C_VEL
LIN {X 0,Y 372.51,Z 1050.437,A -85,B 0,C 180,E1 11080.18,E2 11080.18} C_VEL
LIN {X 0,Y 374.252,Z 1024.481,A -85,B 0,C 180,E1 11087.705,E2 11087.705} C_VEL
LIN {X 0,Y 379.192,Z 985.015,A -85,B 0,C 180,E1 11094.061,E2 11094.061} C_VEL
LIN {X 0,Y 384.866,Z 936.21,A -85,B 0,C 180,E1 11098.401,E2 11098.401} C_VEL
LIN {X 0,Y 387.519,Z 883.62,A -85,B 0,C 180,E1 11100.544,E2 11100.544} C_VEL
LIN {X 0,Y 369.737,Z 831.81,A -85,B 0,C 180,E1 11102.878,E2 11102.878} C_VEL
LIN {X 0,Y 369.414,Z 831.81,A -85,B 0,C 180,E1 11114.03,E2 11114.03} C_VEL
LIN {X 0,Y 369.408,Z 831.81,A -85,B 0,C 180,E1 11123.435,E2 11123.435} C_VEL
LIN {X 0,Y 369.755,Z 831.81,A -85,B 0,C 180,E1 11134.469,E2 11134.469} C_VEL
LIN {X 0,Y 370.369,Z 831.81,A -85,B 0,C 180,E1 11144.551,E2 11144.551} C_VEL
LIN {X 0,Y 370.918,Z 831.81,A -85,B 0,C 180,E1 11154.127,E2 11154.127} C_VEL
LIN {X 0,Y 371.005,Z 831.81,A -85,B 0,C 180,E1 11163.515,E2 11163.515} C_VEL
LIN {X 0,Y 370.405,Z 831.81,A -85,B 0,C 180,E1 11175.443,E2 11175.443} C_VEL
LIN {X 0,Y 369.93,Z 831.81,A -85,B 0,C 180,E1 11185.513,E2 11185.513} C_VEL
LIN {X 0,Y 369.381,Z 831.81,A -85,B 0,C 180,E1 11196.762,E2 11196.762} C_VEL
LIN {X 0,Y 369.357,Z 831.81,A -85,B 0,C 180,E1 11207.318,E2 11207.318} C_VEL
LIN {X 0,Y 369.543,Z 831.81,A -85,B 0,C 180,E1 11219.115,E2 11219.115} C_VEL
LIN {X 0,Y 369.759,Z 831.81,A -85,B 0,C 180,E1 11229.582,E2 11229.582} C_VEL
LIN {X 0,Y 370.674,Z 831.81,A -85,B 0,C 180,E1 11241.761,E2 11241.761} C_VEL
LIN {X 0,Y 371.329,Z 833.326,A -85,B 0,C 180,E1 11248.184,E2 11248.184} C_VEL
LIN {X 0,Y 381.347,Z 876.129,A -85,B 0,C 180,E1 11251.293,E2 11251.293} C_VEL
LIN {X 0,Y 377.941,Z 911.789,A -85,B 0,C 180,E1 11255.472,E2 11255.472} C_VEL
LIN {X 0,Y 374.669,Z 936.734,A -85,B 0,C 180,E1 11261.092,E2 11261.092} C_VEL
LIN {X 0,Y 373.202,Z 949.128,A -85,B 0,C 180,E1 11267.756,E2 11267.756} C_VEL
LIN {X 0,Y 373.894,Z 946.886,A -85,B 0,C 180,E1 11275.224,E2 11275.224} C_VEL
LIN {X 0,Y 376.987,Z 929.866,A -85,B 0,C 180,E1 11281.781,E2 11281.781} C_VEL
LIN {X 0,Y 381.65,Z 900.426,A -85,B 0,C 180,E1 11287.026,E2 11287.026} C_VEL
LIN {X 0,Y 382.483,Z 870.136,A -85,B 0,C 180,E1 11290.203,E2 11290.203} C_VEL
LIN {X 0,Y 369.558,Z 831.81,A -85,B 0,C 180,E1 11293.477,E2 11293.477} C_VEL
LIN {X 0,Y 369.325,Z 831.81,A -85,B 0,C 180,E1 11303.431,E2 11303.431} C_VEL
LIN {X 0,Y 369.697,Z 831.81,A -85,B 0,C 180,E1 11314.47,E2 11314.47} C_VEL
LIN {X 0,Y 370.109,Z 831.81,A -85,B 0,C 180,E1 11324.544,E2 11324.544} C_VEL
LIN {X 0,Y 370.995,Z 831.81,A -85,B 0,C 180,E1 11336.484,E2 11336.484} C_VEL
LIN {X 0,Y 370.801,Z 831.81,A -85,B 0,C 180,E1 11348.238,E2 11348.238} C_VEL
LIN {X 0,Y 370.214,Z 831.81,A -85,B 0,C 180,E1 11357.908,E2 11357.908} C_VEL
LIN {X 0,Y 369.757,Z 831.81,A -85,B 0,C 180,E1 11368.167,E2 11368.167} C_VEL
LIN {X 0,Y 369.442,Z 831.81,A -85,B 0,C 180,E1 11379.551,E2 11379.551} C_VEL
LIN {X 0,Y 369.364,Z 831.81,A -85,B 0,C 180,E1 11390.445,E2 11390.445} C_VEL
LIN {X 0,Y 369.856,Z 833.651,A -85,B 0,C 180,E1 11396.131,E2 11396.131} C_VEL
LIN {X 0,Y 389.961,Z 887.723,A -85,B 0,C 180,E1 11399.051,E2 11399.051} C_VEL
LIN {X 0,Y 385.513,Z 940.866,A -85,B 0,C 180,E1 11401.412,E2 11401.412} C_VEL
LIN {X 0,Y 379.297,Z 988.169,A -85,B 0,C 180,E1 11405.947,E2 11405.947} C_VEL
LIN {X 0,Y 374.352,Z 1026.993,A -85,B 0,C 180,E1 11412.605,E2 11412.605} C_VEL
LIN {X 0,Y 372.349,Z 1052.548,A -85,B 0,C 180,E1 11420.618,E2 11420.618} C_VEL
LIN {X 0,Y 372.413,Z 1061.361,A -85,B 0,C 180,E1 11426.806,E2 11426.806} C_VEL
LIN {X 0,Y 372.489,Z 1059.951,A -85,B 0,C 180,E1 11434.674,E2 11434.674} C_VEL
LIN {X 0,Y 372.51,Z 1050.437,A -85,B 0,C 180,E1 11440.18,E2 11440.18} C_VEL
LIN {X 0,Y 365.28,Z 1035.398,A -85,B 0,C 180,E1 11445.048,E2 11445.048} C_VEL
LIN {X 0,Y 369.327,Z 1000.636,A -85,B 0,C 180,E1 11452.165,E2 11452.165} C_VEL
LIN {X 0,Y 375.244,Z 955.078,A -85,B 0,C 180,E1 11457.407,E2 11457.407} C_VEL
LIN {X 0,Y 380.193,Z 903.493,A -85,B 0,C 180,E1 11460.397,E2 11460.397} C_VEL
LIN {X 0,Y 378.279,Z 879.135,A -85,B 0,C 180,E1 11461.231,E2 11461.231} C_VEL
LIN {X 0,Y 361.68,Z 831.81,A -85,B 0,C 180,E1 11463.468,E2 11463.468} C_VEL
LIN {X 0,Y 361.408,Z 831.81,A -85,B 0,C 180,E1 11473.855,E2 11473.855} C_VEL
LIN {X 0,Y 361.377,Z 831.81,A -85,B 0,C 180,E1 11485.46,E2 11485.46} C_VEL
LIN {X 0,Y 361.821,Z 831.81,A -85,B 0,C 180,E1 11496.515,E2 11496.515} C_VEL
LIN {X 0,Y 362.44,Z 831.81,A -85,B 0,C 180,E1 11506.683,E2 11506.683} C_VEL
LIN {X 0,Y 362.93,Z 831.81,A -85,B 0,C 180,E1 11516.401,E2 11516.401} C_VEL
LIN {X 0,Y 362.791,Z 831.81,A -85,B 0,C 180,E1 11526.001,E2 11526.001} C_VEL
LIN {X 0,Y 362.369,Z 831.81,A -85,B 0,C 180,E1 11535.794,E2 11535.794} C_VEL
LIN {X 0,Y 361.85,Z 831.81,A -85,B 0,C 180,E1 11546.125,E2 11546.125} C_VEL
LIN {X 0,Y 361.289,Z 831.81,A -85,B 0,C 180,E1 11557.521,E2 11557.521} C_VEL
LIN {X 0,Y 361.323,Z 831.81,A -85,B 0,C 180,E1 11569.383,E2 11569.383} C_VEL
LIN {X 0,Y 361.552,Z 831.81,A -85,B 0,C 180,E1 11581.138,E2 11581.138} C_VEL
LIN {X 0,Y 361.848,Z 831.81,A -85,B 0,C 180,E1 11591.667,E2 11591.667} C_VEL
LIN {X 0,Y 362.634,Z 831.81,A -85,B 0,C 180,E1 11601.577,E2 11601.577} C_VEL
LIN {X 0,Y 363.18,Z 832.889,A -85,B 0,C 180,E1 11607.605,E2 11607.605} C_VEL
LIN {X 0,Y 373.56,Z 876.431,A -85,B 0,C 180,E1 11610.806,E2 11610.806} C_VEL
LIN {X 0,Y 370.164,Z 913.615,A -85,B 0,C 180,E1 11615.292,E2 11615.292} C_VEL
LIN {X 0,Y 366.681,Z 939.056,A -85,B 0,C 180,E1 11621.323,E2 11621.323} C_VEL
LIN {X 0,Y 365.258,Z 950.634,A -85,B 0,C 180,E1 11628.155,E2 11628.155} C_VEL
LIN {X 0,Y 366.149,Z 947.512,A -85,B 0,C 180,E1 11635.796,E2 11635.796} C_VEL
LIN {X 0,Y 369.48,Z 930.471,A -85,B 0,C 180,E1 11642.278,E2 11642.278} C_VEL
LIN {X 0,Y 374.582,Z 900.296,A -85,B 0,C 180,E1 11647.66,E2 11647.66} C_VEL
LIN {X 0,Y 375.495,Z 873.087,A -85,B 0,C 180,E1 11650.587,E2 11650.587} C_VEL
LIN {X 0,Y 361.438,Z 831.81,A -85,B 0,C 180,E1 11654.336,E2 11654.336} C_VEL
LIN {X 0,Y 361.322,Z 831.81,A -85,B 0,C 180,E1 11665.46,E2 11665.46} C_VEL
LIN {X 0,Y 361.64,Z 831.81,A -85,B 0,C 180,E1 11676.508,E2 11676.508} C_VEL
LIN {X 0,Y 362.169,Z 831.81,A -85,B 0,C 180,E1 11686.678,E2 11686.678} C_VEL
LIN {X 0,Y 363.429,Z 831.81,A -85,B 0,C 180,E1 11698.806,E2 11698.806} C_VEL
LIN {X 0,Y 362.592,Z 831.81,A -85,B 0,C 180,E1 11710.859,E2 11710.859} C_VEL
LIN {X 0,Y 362.035,Z 831.81,A -85,B 0,C 180,E1 11720.877,E2 11720.877} C_VEL
LIN {X 0,Y 361.59,Z 831.81,A -85,B 0,C 180,E1 11731.647,E2 11731.647} C_VEL
LIN {X 0,Y 361.402,Z 831.81,A -85,B 0,C 180,E1 11743.862,E2 11743.862} C_VEL
LIN {X 0,Y 361.654,Z 832.991,A -85,B 0,C 180,E1 11755.287,E2 11755.287} C_VEL
LIN {X 0,Y 382.777,Z 888.297,A -85,B 0,C 180,E1 11758.481,E2 11758.481} C_VEL
LIN {X 0,Y 378.229,Z 940.498,A -85,B 0,C 180,E1 11760.891,E2 11760.891} C_VEL
LIN {X 0,Y 371.656,Z 988.053,A -85,B 0,C 180,E1 11765.581,E2 11765.581} C_VEL
LIN {X 0,Y 366.493,Z 1025.866,A -85,B 0,C 180,E1 11772.234,E2 11772.234} C_VEL
LIN {X 0,Y 364.436,Z 1051.368,A -85,B 0,C 180,E1 11780.412,E2 11780.412} C_VEL
LIN {X 0,Y 364.497,Z 1059.929,A -85,B 0,C 180,E1 11786.42,E2 11786.42} C_VEL
LIN {X 0,Y 364.604,Z 1059.825,A -85,B 0,C 180,E1 11793.58,E2 11793.58} C_VEL
LIN {X 0,Y 364.451,Z 1046.777,A -85,B 0,C 180,E1 11801.341,E2 11801.341} C_VEL
LIN {X 0,Y 365.28,Z 1035.398,A -85,B 0,C 180,E1 11805.048,E2 11805.048} C_VEL
LIN {X 0,Y 359.124,Z 1015.845,A -85,B 0,C 180,E1 11809.646,E2 11809.646} C_VEL
LIN {X 0,Y 365.009,Z 974.328,A -85,B 0,C 180,E1 11815.884,E2 11815.884} C_VEL
LIN {X 0,Y 371.048,Z 924.755,A -85,B 0,C 180,E1 11819.898,E2 11819.898} C_VEL
LIN {X 0,Y 371.759,Z 883.634,A -85,B 0,C 180,E1 11821.561,E2 11821.561} C_VEL
LIN {X 0,Y 353.606,Z 831.81,A -85,B 0,C 180,E1 11824.137,E2 11824.137} C_VEL
LIN {X 0,Y 353.336,Z 831.81,A -85,B 0,C 180,E1 11835.126,E2 11835.126} C_VEL
LIN {X 0,Y 353.367,Z 831.81,A -85,B 0,C 180,E1 11847.528,E2 11847.528} C_VEL
LIN {X 0,Y 353.891,Z 831.81,A -85,B 0,C 180,E1 11858.62,E2 11858.62} C_VEL
LIN {X 0,Y 354.541,Z 831.81,A -85,B 0,C 180,E1 11868.892,E2 11868.892} C_VEL
LIN {X 0,Y 355.441,Z 831.81,A -85,B 0,C 180,E1 11881.221,E2 11881.221} C_VEL
LIN {X 0,Y 354.406,Z 831.81,A -85,B 0,C 180,E1 11893.62,E2 11893.62} C_VEL
LIN {X 0,Y 353.893,Z 831.81,A -85,B 0,C 180,E1 11904.039,E2 11904.039} C_VEL
LIN {X 0,Y 353.311,Z 831.81,A -85,B 0,C 180,E1 11915.44,E2 11915.44} C_VEL
LIN {X 0,Y 353.285,Z 831.81,A -85,B 0,C 180,E1 11925.134,E2 11925.134} C_VEL
LIN {X 0,Y 353.364,Z 831.81,A -85,B 0,C 180,E1 11937.532,E2 11937.532} C_VEL
LIN {X 0,Y 353.653,Z 831.81,A -85,B 0,C 180,E1 11948.608,E2 11948.608} C_VEL
LIN {X 0,Y 354.391,Z 831.81,A -85,B 0,C 180,E1 11958.889,E2 11958.889} C_VEL
LIN {X 0,Y 355.207,Z 833.328,A -85,B 0,C 180,E1 11967.034,E2 11967.034} C_VEL
LIN {X 0,Y 365.824,Z 877.094,A -85,B 0,C 180,E1 11970.344,E2 11970.344} C_VEL
LIN {X 0,Y 362.681,Z 913.611,A -85,B 0,C 180,E1 11974.8,E2 11974.8} C_VEL
LIN {X 0,Y 358.918,Z 939.654,A -85,B 0,C 180,E1 11980.968,E2 11980.968} C_VEL
LIN {X 0,Y 357.45,Z 951.08,A -85,B 0,C 180,E1 11987.207,E2 11987.207} C_VEL
LIN {X 0,Y 357.938,Z 950.833,A -85,B 0,C 180,E1 11994.281,E2 11994.281} C_VEL
LIN {X 0,Y 361.061,Z 936.498,A -85,B 0,C 180,E1 12001.281,E2 12001.281} C_VEL
LIN {X 0,Y 366.187,Z 908.632,A -85,B 0,C 180,E1 12007.15,E2 12007.15} C_VEL
LIN {X 0,Y 368.511,Z 876.119,A -85,B 0,C 180,E1 12010.966,E2 12010.966} C_VEL
LIN {X 0,Y 354.582,Z 836.049,A -85,B 0,C 180,E1 12014.862,E2 12014.862} C_VEL
LIN {X 0,Y 353.324,Z 831.81,A -85,B 0,C 180,E1 12015.615,E2 12015.615} C_VEL
LIN {X 0,Y 353.334,Z 831.81,A -85,B 0,C 180,E1 12027.53,E2 12027.53} C_VEL
LIN {X 0,Y 353.644,Z 831.81,A -85,B 0,C 180,E1 12038.609,E2 12038.609} C_VEL
LIN {X 0,Y 354.395,Z 831.81,A -85,B 0,C 180,E1 12048.892,E2 12048.892} C_VEL
LIN {X 0,Y 355.436,Z 831.81,A -85,B 0,C 180,E1 12058.779,E2 12058.779} C_VEL
LIN {X 0,Y 354.545,Z 831.81,A -85,B 0,C 180,E1 12071.108,E2 12071.108} C_VEL
LIN {X 0,Y 353.896,Z 831.81,A -85,B 0,C 180,E1 12082.79,E2 12082.79} C_VEL
LIN {X 0,Y 353.433,Z 831.81,A -85,B 0,C 180,E1 12093.148,E2 12093.148} C_VEL
LIN {X 0,Y 353.331,Z 831.81,A -85,B 0,C 180,E1 12105.133,E2 12105.133} C_VEL
LIN {X 0,Y 353.646,Z 833.568,A -85,B 0,C 180,E1 12114.446,E2 12114.446} C_VEL
LIN {X 0,Y 375.373,Z 888.394,A -85,B 0,C 180,E1 12117.854,E2 12117.854} C_VEL
LIN {X 0,Y 370.888,Z 941.248,A -85,B 0,C 180,E1 12120.426,E2 12120.426} C_VEL
LIN {X 0,Y 364.039,Z 987.937,A -85,B 0,C 180,E1 12125.2,E2 12125.2} C_VEL
LIN {X 0,Y 358.586,Z 1025.342,A -85,B 0,C 180,E1 12131.989,E2 12131.989} C_VEL
LIN {X 0,Y 356.503,Z 1050.191,A -85,B 0,C 180,E1 12140.197,E2 12140.197} C_VEL
LIN {X 0,Y 356.805,Z 1059.888,A -85,B 0,C 180,E1 12148.357,E2 12148.357} C_VEL
LIN {X 0,Y 356.438,Z 1055.974,A -85,B 0,C 180,E1 12156.11,E2 12156.11} C_VEL
LIN {X 0,Y 356.879,Z 1038.06,A -85,B 0,C 180,E1 12164.153,E2 12164.153} C_VEL
LIN {X 0,Y 359.124,Z 1015.845,A -85,B 0,C 180,E1 12169.646,E2 12169.646} C_VEL
LIN {X 0,Y 354.769,Z 992.302,A -85,B 0,C 180,E1 12173.866,E2 12173.866} C_VEL
LIN {X 0,Y 361.088,Z 946.246,A -85,B 0,C 180,E1 12178.902,E2 12178.902} C_VEL
LIN {X 0,Y 365.937,Z 894.007,A -85,B 0,C 180,E1 12181.651,E2 12181.651} C_VEL
LIN {X 0,Y 345.523,Z 831.81,A -85,B 0,C 180,E1 12184.603,E2 12184.603} C_VEL
LIN {X 0,Y 345.22,Z 831.81,A -85,B 0,C 180,E1 12197.043,E2 12197.043} C_VEL
LIN {X 0,Y 345.34,Z 831.81,A -85,B 0,C 180,E1 12208.971,E2 12208.971} C_VEL
LIN {X 0,Y 345.98,Z 831.81,A -85,B 0,C 180,E1 12220.79,E2 12220.79} C_VEL
LIN {X 0,Y 346.684,Z 831.81,A -85,B 0,C 180,E1 12231.184,E2 12231.184} C_VEL
LIN {X 0,Y 347.422,Z 831.81,A -85,B 0,C 180,E1 12241.249,E2 12241.249} C_VEL
LIN {X 0,Y 346.386,Z 831.81,A -85,B 0,C 180,E1 12253.941,E2 12253.941} C_VEL
LIN {X 0,Y 345.697,Z 831.81,A -85,B 0,C 180,E1 12265.853,E2 12265.853} C_VEL
LIN {X 0,Y 345.274,Z 831.81,A -85,B 0,C 180,E1 12276.394,E2 12276.394} C_VEL
LIN {X 0,Y 345.166,Z 831.81,A -85,B 0,C 180,E1 12287.041,E2 12287.041} C_VEL
LIN {X 0,Y 345.338,Z 831.81,A -85,B 0,C 180,E1 12298.971,E2 12298.971} C_VEL
LIN {X 0,Y 345.736,Z 831.81,A -85,B 0,C 180,E1 12310.779,E2 12310.779} C_VEL
LIN {X 0,Y 346.556,Z 831.81,A -85,B 0,C 180,E1 12321.184,E2 12321.184} C_VEL
LIN {X 0,Y 347.178,Z 833.606,A -85,B 0,C 180,E1 12326.427,E2 12326.427} C_VEL
LIN {X 0,Y 357.842,Z 876.382,A -85,B 0,C 180,E1 12329.724,E2 12329.724} C_VEL
LIN {X 0,Y 355.554,Z 911.603,A -85,B 0,C 180,E1 12333.977,E2 12333.977} C_VEL
LIN {X 0,Y 351.497,Z 938.285,A -85,B 0,C 180,E1 12339.944,E2 12339.944} C_VEL
LIN {X 0,Y 349.642,Z 951.439,A -85,B 0,C 180,E1 12346.386,E2 12346.386} C_VEL
LIN {X 0,Y 350.061,Z 952.162,A -85,B 0,C 180,E1 12354.319,E2 12354.319} C_VEL
LIN {X 0,Y 353.496,Z 937.44,A -85,B 0,C 180,E1 12361.713,E2 12361.713} C_VEL
LIN {X 0,Y 358.897,Z 909.845,A -85,B 0,C 180,E1 12367.631,E2 12367.631} C_VEL
LIN {X 0,Y 361.494,Z 878.712,A -85,B 0,C 180,E1 12371.418,E2 12371.418} C_VEL
LIN {X 0,Y 347.652,Z 838.036,A -85,B 0,C 180,E1 12375.582,E2 12375.582} C_VEL
LIN {X 0,Y 345.285,Z 831.81,A -85,B 0,C 180,E1 12376.483,E2 12376.483} C_VEL
LIN {X 0,Y 345.314,Z 831.81,A -85,B 0,C 180,E1 12388.976,E2 12388.976} C_VEL
LIN {X 0,Y 345.726,Z 831.81,A -85,B 0,C 180,E1 12400.781,E2 12400.781} C_VEL
LIN {X 0,Y 346.561,Z 831.81,A -85,B 0,C 180,E1 12411.186,E2 12411.186} C_VEL
LIN {X 0,Y 347.017,Z 831.81,A -85,B 0,C 180,E1 12421.255,E2 12421.255} C_VEL
LIN {X 0,Y 346.511,Z 831.81,A -85,B 0,C 180,E1 12431.369,E2 12431.369} C_VEL
LIN {X 0,Y 345.912,Z 831.81,A -85,B 0,C 180,E1 12441.899,E2 12441.899} C_VEL
LIN {X 0,Y 345.412,Z 831.81,A -85,B 0,C 180,E1 12453.316,E2 12453.316} C_VEL
LIN {X 0,Y 345.236,Z 831.81,A -85,B 0,C 180,E1 12463.508,E2 12463.508} C_VEL
LIN {X 0,Y 345.461,Z 833.107,A -85,B 0,C 180,E1 12473.498,E2 12473.498} C_VEL
LIN {X 0,Y 367.927,Z 888.366,A -85,B 0,C 180,E1 12477.19,E2 12477.19} C_VEL
LIN {X 0,Y 363.876,Z 940.052,A -85,B 0,C 180,E1 12479.798,E2 12479.798} C_VEL
LIN {X 0,Y 356.626,Z 986.837,A -85,B 0,C 180,E1 12484.648,E2 12484.648} C_VEL
LIN {X 0,Y 350.705,Z 1024.165,A -85,B 0,C 180,E1 12491.569,E2 12491.569} C_VEL
LIN {X 0,Y 348.551,Z 1049.036,A -85,B 0,C 180,E1 12499.971,E2 12499.971} C_VEL
LIN {X 0,Y 348.671,Z 1057.574,A -85,B 0,C 180,E1 12506.257,E2 12506.257} C_VEL
LIN {X 0,Y 348.77,Z 1057.36,A -85,B 0,C 180,E1 12513.743,E2 12513.743} C_VEL
LIN {X 0,Y 348.544,Z 1043.953,A -85,B 0,C 180,E1 12521.876,E2 12521.876} C_VEL
LIN {X 0,Y 351.05,Z 1016.697,A -85,B 0,C 180,E1 12529.574,E2 12529.574} C_VEL
LIN {X 0,Y 354.769,Z 992.302,A -85,B 0,C 180,E1 12533.866,E2 12533.866} C_VEL
LIN {X 0,Y 350.868,Z 965.274,A -85,B 0,C 180,E1 12537.548,E2 12537.548} C_VEL
LIN {X 0,Y 357.069,Z 915.141,A -85,B 0,C 180,E1 12541.304,E2 12541.304} C_VEL
LIN {X 0,Y 356.596,Z 885.425,A -85,B 0,C 180,E1 12542.555,E2 12542.555} C_VEL
LIN {X 0,Y 337.46,Z 831.81,A -85,B 0,C 180,E1 12545.285,E2 12545.285} C_VEL
LIN {X 0,Y 337.119,Z 831.81,A -85,B 0,C 180,E1 12557.967,E2 12557.967} C_VEL
LIN {X 0,Y 337.33,Z 831.81,A -85,B 0,C 180,E1 12568.84,E2 12568.84} C_VEL
LIN {X 0,Y 337.924,Z 831.81,A -85,B 0,C 180,E1 12580.314,E2 12580.314} C_VEL
LIN {X 0,Y 338.657,Z 831.81,A -85,B 0,C 180,E1 12590.974,E2 12590.974} C_VEL
LIN {X 0,Y 339.408,Z 831.81,A -85,B 0,C 180,E1 12601.279,E2 12601.279} C_VEL
LIN {X 0,Y 338.494,Z 831.81,A -85,B 0,C 180,E1 12611.637,E2 12611.637} C_VEL
LIN {X 0,Y 337.808,Z 831.81,A -85,B 0,C 180,E1 12622.938,E2 12622.938} C_VEL
LIN {X 0,Y 337.29,Z 831.81,A -85,B 0,C 180,E1 12634.221,E2 12634.221} C_VEL
LIN {X 0,Y 337.088,Z 831.81,A -85,B 0,C 180,E1 12645.749,E2 12645.749} C_VEL
LIN {X 0,Y 337.297,Z 831.81,A -85,B 0,C 180,E1 12656.34,E2 12656.34} C_VEL
LIN {X 0,Y 337.557,Z 831.81,A -85,B 0,C 180,E1 12667.534,E2 12667.534} C_VEL
LIN {X 0,Y 338.274,Z 831.81,A -85,B 0,C 180,E1 12678.353,E2 12678.353} C_VEL
LIN {X 0,Y 339.057,Z 833.66,A -85,B 0,C 180,E1 12685.788,E2 12685.788} C_VEL
LIN {X 0,Y 349.64,Z 874.246,A -85,B 0,C 180,E1 12688.936,E2 12688.936} C_VEL
LIN {X 0,Y 349.85,Z 899.577,A -85,B 0,C 180,E1 12691.738,E2 12691.738} C_VEL
LIN {X 0,Y 345.103,Z 931.34,A -85,B 0,C 180,E1 12697.426,E2 12697.426} C_VEL
LIN {X 0,Y 342.229,Z 949.538,A -85,B 0,C 180,E1 12704.115,E2 12704.115} C_VEL
LIN {X 0,Y 341.706,Z 954.79,A -85,B 0,C 180,E1 12712.178,E2 12712.178} C_VEL
LIN {X 0,Y 344.194,Z 945.07,A -85,B 0,C 180,E1 12719.736,E2 12719.736} C_VEL
LIN {X 0,Y 349.465,Z 921.238,A -85,B 0,C 180,E1 12726.391,E2 12726.391} C_VEL
LIN {X 0,Y 355.178,Z 885.395,A -85,B 0,C 180,E1 12731.377,E2 12731.377} C_VEL
LIN {X 0,Y 343.225,Z 845.786,A -85,B 0,C 180,E1 12735.789,E2 12735.789} C_VEL
LIN {X 0,Y 337.202,Z 831.81,A -85,B 0,C 180,E1 12737.223,E2 12737.223} C_VEL
LIN {X 0,Y 337.303,Z 831.81,A -85,B 0,C 180,E1 12748.844,E2 12748.844} C_VEL
LIN {X 0,Y 337.693,Z 831.81,A -85,B 0,C 180,E1 12760.305,E2 12760.305} C_VEL
LIN {X 0,Y 338.543,Z 831.81,A -85,B 0,C 180,E1 12770.976,E2 12770.976} C_VEL
LIN {X 0,Y 339.023,Z 831.81,A -85,B 0,C 180,E1 12781.285,E2 12781.285} C_VEL
LIN {X 0,Y 338.46,Z 831.81,A -85,B 0,C 180,E1 12791.643,E2 12791.643} C_VEL
LIN {X 0,Y 337.774,Z 831.81,A -85,B 0,C 180,E1 12802.926,E2 12802.926} C_VEL
LIN {X 0,Y 337.354,Z 831.81,A -85,B 0,C 180,E1 12814.22,E2 12814.22} C_VEL
LIN {X 0,Y 337.141,Z 831.81,A -85,B 0,C 180,E1 12825.759,E2 12825.759} C_VEL
LIN {X 0,Y 337.365,Z 832.847,A -85,B 0,C 180,E1 12832.498,E2 12832.498} C_VEL
LIN {X 0,Y 360.833,Z 889.341,A -85,B 0,C 180,E1 12836.548,E2 12836.548} C_VEL
LIN {X 0,Y 356.593,Z 940.802,A -85,B 0,C 180,E1 12839.291,E2 12839.291} C_VEL
LIN {X 0,Y 348.83,Z 987.909,A -85,B 0,C 180,E1 12844.386,E2 12844.386} C_VEL
LIN {X 0,Y 342.688,Z 1024.816,A -85,B 0,C 180,E1 12851.591,E2 12851.591} C_VEL
LIN {X 0,Y 340.548,Z 1049.133,A -85,B 0,C 180,E1 12860.381,E2 12860.381} C_VEL
LIN {X 0,Y 341.094,Z 1057.602,A -85,B 0,C 180,E1 12868.726,E2 12868.726} C_VEL
LIN {X 0,Y 340.556,Z 1053.401,A -85,B 0,C 180,E1 12876.397,E2 12876.397} C_VEL
LIN {X 0,Y 341.184,Z 1035.084,A -85,B 0,C 180,E1 12884.819,E2 12884.819} C_VEL
LIN {X 0,Y 345.396,Z 1002.26,A -85,B 0,C 180,E1 12892.493,E2 12892.493} C_VEL
LIN {X 0,Y 350.868,Z 965.274,A -85,B 0,C 180,E1 12897.548,E2 12897.548} C_VEL
LIN {X 0,Y 347.377,Z 935.185,A -85,B 0,C 180,E1 12900.585,E2 12900.585} C_VEL
LIN {X 0,Y 349.637,Z 888.452,A -85,B 0,C 180,E1 12902.968,E2 12902.968} C_VEL
LIN {X 0,Y 329.406,Z 831.81,A -85,B 0,C 180,E1 12906.264,E2 12906.264} C_VEL
LIN {X 0,Y 329.115,Z 831.81,A -85,B 0,C 180,E1 12918.035,E2 12918.035} C_VEL
LIN {X 0,Y 329.319,Z 831.81,A -85,B 0,C 180,E1 12928.486,E2 12928.486} C_VEL
LIN {X 0,Y 329.911,Z 831.81,A -85,B 0,C 180,E1 12940.557,E2 12940.557} C_VEL
LIN {X 0,Y 330.8,Z 831.81,A -85,B 0,C 180,E1 12953.411,E2 12953.411} C_VEL
LIN {X 0,Y 330.911,Z 831.81,A -85,B 0,C 180,E1 12963.942,E2 12963.942} C_VEL
LIN {X 0,Y 330.303,Z 831.81,A -85,B 0,C 180,E1 12974.635,E2 12974.635} C_VEL
LIN {X 0,Y 329.607,Z 831.81,A -85,B 0,C 180,E1 12986.129,E2 12986.129} C_VEL
LIN {X 0,Y 329.062,Z 831.81,A -85,B 0,C 180,E1 12998.504,E2 12998.504} C_VEL
LIN {X 0,Y 329.027,Z 831.81,A -85,B 0,C 180,E1 13009.554,E2 13009.554} C_VEL
LIN {X 0,Y 329.356,Z 831.81,A -85,B 0,C 180,E1 13021.066,E2 13021.066} C_VEL
LIN {X 0,Y 329.756,Z 831.81,A -85,B 0,C 180,E1 13032.594,E2 13032.594} C_VEL
LIN {X 0,Y 330.794,Z 832.481,A -85,B 0,C 180,E1 13045.065,E2 13045.065} C_VEL
LIN {X 0,Y 341.618,Z 873.019,A -85,B 0,C 180,E1 13048.213,E2 13048.213} C_VEL
LIN {X 0,Y 342.517,Z 898.881,A -85,B 0,C 180,E1 13051.11,E2 13051.11} C_VEL
LIN {X 0,Y 337.527,Z 931.109,A -85,B 0,C 180,E1 13056.809,E2 13056.809} C_VEL
LIN {X 0,Y 334.468,Z 949.855,A -85,B 0,C 180,E1 13063.536,E2 13063.536} C_VEL
LIN {X 0,Y 333.685,Z 956.205,A -85,B 0,C 180,E1 13071.201,E2 13071.201} C_VEL
LIN {X 0,Y 335.926,Z 948.461,A -85,B 0,C 180,E1 13079.053,E2 13079.053} C_VEL
LIN {X 0,Y 341.25,Z 926.221,A -85,B 0,C 180,E1 13086.112,E2 13086.112} C_VEL
LIN {X 0,Y 348.044,Z 891.273,A -85,B 0,C 180,E1 13091.446,E2 13091.446} C_VEL
LIN {X 0,Y 339.02,Z 854.29,A -85,B 0,C 180,E1 13095.844,E2 13095.844} C_VEL
LIN {X 0,Y 329.069,Z 831.81,A -85,B 0,C 180,E1 13098.443,E2 13098.443} C_VEL
LIN {X 0,Y 329.338,Z 831.81,A -85,B 0,C 180,E1 13111.066,E2 13111.066} C_VEL
LIN {X 0,Y 329.781,Z 831.81,A -85,B 0,C 180,E1 13122.598,E2 13122.598} C_VEL
LIN {X 0,Y 330.625,Z 831.81,A -85,B 0,C 180,E1 13133.413,E2 13133.413} C_VEL
LIN {X 0,Y 331.015,Z 831.81,A -85,B 0,C 180,E1 13141.316,E2 13141.316} C_VEL
LIN {X 0,Y 330.409,Z 831.81,A -85,B 0,C 180,E1 13151.931,E2 13151.931} C_VEL
LIN {X 0,Y 329.772,Z 831.81,A -85,B 0,C 180,E1 13163.031,E2 13163.031} C_VEL
LIN {X 0,Y 329.208,Z 831.81,A -85,B 0,C 180,E1 13175.19,E2 13175.19} C_VEL
LIN {X 0,Y 329.133,Z 831.81,A -85,B 0,C 180,E1 13185.623,E2 13185.623} C_VEL
LIN {X 0,Y 329.22,Z 832.415,A -85,B 0,C 180,E1 13191.422,E2 13191.422} C_VEL
LIN {X 0,Y 353.634,Z 889.819,A -85,B 0,C 180,E1 13195.843,E2 13195.843} C_VEL
LIN {X 0,Y 349.994,Z 937.843,A -85,B 0,C 180,E1 13198.466,E2 13198.466} C_VEL
LIN {X 0,Y 341.859,Z 984.63,A -85,B 0,C 180,E1 13203.47,E2 13203.47} C_VEL
LIN {X 0,Y 335.089,Z 1021.634,A -85,B 0,C 180,E1 13210.601,E2 13210.601} C_VEL
LIN {X 0,Y 332.722,Z 1045.272,A -85,B 0,C 180,E1 13218.729,E2 13218.729} C_VEL
LIN {X 0,Y 332.82,Z 1055.232,A -85,B 0,C 180,E1 13226.079,E2 13226.079} C_VEL
LIN {X 0,Y 332.898,Z 1054.867,A -85,B 0,C 180,E1 13233.921,E2 13233.921} C_VEL
LIN {X 0,Y 332.614,Z 1040.941,A -85,B 0,C 180,E1 13242.517,E2 13242.517} C_VEL
LIN {X 0,Y 335.549,Z 1013.245,A -85,B 0,C 180,E1 13250.518,E2 13250.518} C_VEL
LIN {X 0,Y 341.996,Z 972.829,A -85,B 0,C 180,E1 13257.054,E2 13257.054} C_VEL
LIN {X 0,Y 347.377,Z 935.185,A -85,B 0,C 180,E1 13260.585,E2 13260.585} C_VEL
LIN {X 0,Y 343.396,Z 902.719,A -85,B 0,C 180,E1 13262.876,E2 13262.876} C_VEL
LIN {X 0,Y 336.845,Z 873.5,A -85,B 0,C 180,E1 13264.335,E2 13264.335} C_VEL
LIN {X 0,Y 321.33,Z 831.81,A -85,B 0,C 180,E1 13266.689,E2 13266.689} C_VEL
LIN {X 0,Y 321.055,Z 831.81,A -85,B 0,C 180,E1 13277.109,E2 13277.109} C_VEL
LIN {X 0,Y 321.135,Z 831.81,A -85,B 0,C 180,E1 13287.077,E2 13287.077} C_VEL
LIN {X 0,Y 321.742,Z 831.81,A -85,B 0,C 180,E1 13299.279,E2 13299.279} C_VEL
LIN {X 0,Y 322.589,Z 831.81,A -85,B 0,C 180,E1 13310.52,E2 13310.52} C_VEL
LIN {X 0,Y 323.376,Z 831.81,A -85,B 0,C 180,E1 13321.342,E2 13321.342} C_VEL
LIN {X 0,Y 322.385,Z 831.81,A -85,B 0,C 180,E1 13332.227,E2 13332.227} C_VEL
LIN {X 0,Y 321.692,Z 831.81,A -85,B 0,C 180,E1 13343.638,E2 13343.638} C_VEL
LIN {X 0,Y 321.091,Z 831.81,A -85,B 0,C 180,E1 13356.211,E2 13356.211} C_VEL
LIN {X 0,Y 321.002,Z 831.81,A -85,B 0,C 180,E1 13367.118,E2 13367.118} C_VEL
LIN {X 0,Y 321.123,Z 831.81,A -85,B 0,C 180,E1 13377.08,E2 13377.08} C_VEL
LIN {X 0,Y 321.523,Z 831.81,A -85,B 0,C 180,E1 13389.268,E2 13389.268} C_VEL
LIN {X 0,Y 322.43,Z 831.81,A -85,B 0,C 180,E1 13400.518,E2 13400.518} C_VEL
LIN {X 0,Y 322.857,Z 833.359,A -85,B 0,C 180,E1 13404.394,E2 13404.394} C_VEL
LIN {X 0,Y 333.87,Z 872.855,A -85,B 0,C 180,E1 13407.589,E2 13407.589} C_VEL
LIN {X 0,Y 335.165,Z 898.482,A -85,B 0,C 180,E1 13410.504,E2 13410.504} C_VEL
LIN {X 0,Y 329.896,Z 931.188,A -85,B 0,C 180,E1 13416.272,E2 13416.272} C_VEL
LIN {X 0,Y 326.646,Z 950.574,A -85,B 0,C 180,E1 13423.182,E2 13423.182} C_VEL
LIN {X 0,Y 325.702,Z 957.401,A -85,B 0,C 180,E1 13430.453,E2 13430.453} C_VEL
LIN {X 0,Y 327.846,Z 951.112,A -85,B 0,C 180,E1 13438.609,E2 13438.609} C_VEL
LIN {X 0,Y 333.148,Z 930.673,A -85,B 0,C 180,E1 13445.859,E2 13445.859} C_VEL
LIN {X 0,Y 340.323,Z 897.269,A -85,B 0,C 180,E1 13451.511,E2 13451.511} C_VEL
LIN {X 0,Y 335.943,Z 867.455,A -85,B 0,C 180,E1 13455.295,E2 13455.295} C_VEL
LIN {X 0,Y 321.04,Z 831.81,A -85,B 0,C 180,E1 13459.345,E2 13459.345} C_VEL
LIN {X 0,Y 321.325,Z 831.81,A -85,B 0,C 180,E1 13470.891,E2 13470.891} C_VEL
LIN {X 0,Y 321.743,Z 831.81,A -85,B 0,C 180,E1 13482.148,E2 13482.148} C_VEL
LIN {X 0,Y 322.595,Z 831.81,A -85,B 0,C 180,E1 13493.248,E2 13493.248} C_VEL
LIN {X 0,Y 323.022,Z 831.81,A -85,B 0,C 180,E1 13501.349,E2 13501.349} C_VEL
LIN {X 0,Y 322.355,Z 831.81,A -85,B 0,C 180,E1 13512.234,E2 13512.234} C_VEL
LIN {X 0,Y 321.66,Z 831.81,A -85,B 0,C 180,E1 13523.646,E2 13523.646} C_VEL
LIN {X 0,Y 321.179,Z 831.81,A -85,B 0,C 180,E1 13536.206,E2 13536.206} C_VEL
LIN {X 0,Y 321.088,Z 831.81,A -85,B 0,C 180,E1 13548.412,E2 13548.412} C_VEL
LIN {X 0,Y 321.334,Z 833.666,A -85,B 0,C 180,E1 13550.335,E2 13550.335} C_VEL
LIN {X 0,Y 345.557,Z 887.037,A -85,B 0,C 180,E1 13554.887,E2 13554.887} C_VEL
LIN {X 0,Y 346.963,Z 908.989,A -85,B 0,C 180,E1 13556.065,E2 13556.065} C_VEL
LIN {X 0,Y 339.264,Z 959.351,A -85,B 0,C 180,E1 13559.788,E2 13559.788} C_VEL
LIN {X 0,Y 330.851,Z 1001.658,A -85,B 0,C 180,E1 13565.877,E2 13565.877} C_VEL
LIN {X 0,Y 325.66,Z 1032.761,A -85,B 0,C 180,E1 13573.779,E2 13573.779} C_VEL
LIN {X 0,Y 324.586,Z 1049.942,A -85,B 0,C 180,E1 13581.938,E2 13581.938} C_VEL
LIN {X 0,Y 325.244,Z 1055.211,A -85,B 0,C 180,E1 13588.664,E2 13588.664} C_VEL
LIN {X 0,Y 324.701,Z 1050.816,A -85,B 0,C 180,E1 13596.71,E2 13596.71} C_VEL
LIN {X 0,Y 325.74,Z 1031.138,A -85,B 0,C 180,E1 13605.852,E2 13605.852} C_VEL
LIN {X 0,Y 330.303,Z 998.021,A -85,B 0,C 180,E1 13613.661,E2 13613.661} C_VEL
LIN {X 0,Y 337.287,Z 953.989,A -85,B 0,C 180,E1 13619.48,E2 13619.48} C_VEL
LIN {X 0,Y 343.396,Z 902.719,A -85,B 0,C 180,E1 13622.876,E2 13622.876} C_VEL
LIN {X 0,Y 332.391,Z 883.493,A -85,B 0,C 180,E1 13624.441,E2 13624.441} C_VEL
LIN {X 0,Y 313.229,Z 831.81,A -85,B 0,C 180,E1 13627.6,E2 13627.6} C_VEL
LIN {X 0,Y 312.932,Z 831.81,A -85,B 0,C 180,E1 13639.099,E2 13639.099} C_VEL
LIN {X 0,Y 313.156,Z 831.81,A -85,B 0,C 180,E1 13649.409,E2 13649.409} C_VEL
LIN {X 0,Y 313.874,Z 831.81,A -85,B 0,C 180,E1 13661.679,E2 13661.679} C_VEL
LIN {X 0,Y 314.729,Z 831.81,A -85,B 0,C 180,E1 13673.073,E2 13673.073} C_VEL
LIN {X 0,Y 314.865,Z 831.81,A -85,B 0,C 180,E1 13684.143,E2 13684.143} C_VEL
LIN {X 0,Y 314.196,Z 831.81,A -85,B 0,C 180,E1 13695.403,E2 13695.403} C_VEL
LIN {X 0,Y 313.453,Z 831.81,A -85,B 0,C 180,E1 13707.381,E2 13707.381} C_VEL
LIN {X 0,Y 312.998,Z 831.81,A -85,B 0,C 180,E1 13717.304,E2 13717.304} C_VEL
LIN {X 0,Y 312.884,Z 831.81,A -85,B 0,C 180,E1 13729.097,E2 13729.097} C_VEL
LIN {X 0,Y 313.142,Z 831.81,A -85,B 0,C 180,E1 13739.412,E2 13739.412} C_VEL
LIN {X 0,Y 313.63,Z 831.81,A -85,B 0,C 180,E1 13751.668,E2 13751.668} C_VEL
LIN {X 0,Y 314.752,Z 833.137,A -85,B 0,C 180,E1 13763.649,E2 13763.649} C_VEL
LIN {X 0,Y 326.185,Z 872.73,A -85,B 0,C 180,E1 13766.94,E2 13766.94} C_VEL
LIN {X 0,Y 327.725,Z 899.046,A -85,B 0,C 180,E1 13770,E2 13770} C_VEL
LIN {X 0,Y 322.317,Z 931.359,A -85,B 0,C 180,E1 13775.742,E2 13775.742} C_VEL
LIN {X 0,Y 318.899,Z 951.079,A -85,B 0,C 180,E1 13782.698,E2 13782.698} C_VEL
LIN {X 0,Y 317.837,Z 958.637,A -85,B 0,C 180,E1 13790.983,E2 13790.983} C_VEL
LIN {X 0,Y 320.013,Z 952.719,A -85,B 0,C 180,E1 13798.682,E2 13798.682} C_VEL
LIN {X 0,Y 325.779,Z 931.993,A -85,B 0,C 180,E1 13806.338,E2 13806.338} C_VEL
LIN {X 0,Y 333.246,Z 899.369,A -85,B 0,C 180,E1 13812.049,E2 13812.049} C_VEL
LIN {X 0,Y 329.115,Z 869.882,A -85,B 0,C 180,E1 13815.966,E2 13815.966} C_VEL
LIN {X 0,Y 312.997,Z 831.81,A -85,B 0,C 180,E1 13820.813,E2 13820.813} C_VEL
LIN {X 0,Y 313.334,Z 831.81,A -85,B 0,C 180,E1 13833.635,E2 13833.635} C_VEL
LIN {X 0,Y 313.884,Z 831.81,A -85,B 0,C 180,E1 13844.581,E2 13844.581} C_VEL
LIN {X 0,Y 314.831,Z 831.81,A -85,B 0,C 180,E1 13855.856,E2 13855.856} C_VEL
LIN {X 0,Y 314.729,Z 831.81,A -85,B 0,C 180,E1 13866.927,E2 13866.927} C_VEL
LIN {X 0,Y 313.816,Z 831.81,A -85,B 0,C 180,E1 13879.445,E2 13879.445} C_VEL
LIN {X 0,Y 313.169,Z 831.81,A -85,B 0,C 180,E1 13892.005,E2 13892.005} C_VEL
LIN {X 0,Y 312.945,Z 831.81,A -85,B 0,C 180,E1 13904.687,E2 13904.687} C_VEL
LIN {X 0,Y 313.264,Z 833.443,A -85,B 0,C 180,E1 13909.101,E2 13909.101} C_VEL
LIN {X 0,Y 338.396,Z 887.699,A -85,B 0,C 180,E1 13914.095,E2 13914.095} C_VEL
LIN {X 0,Y 340.218,Z 908.791,A -85,B 0,C 180,E1 13915.349,E2 13915.349} C_VEL
LIN {X 0,Y 332.255,Z 958.352,A -85,B 0,C 180,E1 13919.081,E2 13919.081} C_VEL
LIN {X 0,Y 323.288,Z 1001.121,A -85,B 0,C 180,E1 13925.38,E2 13925.38} C_VEL
LIN {X 0,Y 317.789,Z 1031.967,A -85,B 0,C 180,E1 13933.48,E2 13933.48} C_VEL
LIN {X 0,Y 316.658,Z 1048.799,A -85,B 0,C 180,E1 13941.734,E2 13941.734} C_VEL
LIN {X 0,Y 317.311,Z 1054.017,A -85,B 0,C 180,E1 13948.63,E2 13948.63} C_VEL
LIN {X 0,Y 316.774,Z 1049.502,A -85,B 0,C 180,E1 13956.879,E2 13956.879} C_VEL
LIN {X 0,Y 317.777,Z 1030.728,A -85,B 0,C 180,E1 13965.872,E2 13965.872} C_VEL
LIN {X 0,Y 322.485,Z 997.731,A -85,B 0,C 180,E1 13973.946,E2 13973.946} C_VEL
LIN {X 0,Y 329.619,Z 954.51,A -85,B 0,C 180,E1 13979.855,E2 13979.855} C_VEL
LIN {X 0,Y 336.039,Z 902.935,A -85,B 0,C 180,E1 13983.399,E2 13983.399} C_VEL
LIN {X 0,Y 332.391,Z 883.493,A -85,B 0,C 180,E1 13984.441,E2 13984.441} C_VEL
LIN {X 0,Y 314.383,Z 855.526,A -85,B 0,C 180,E1 13986.689,E2 13986.689} C_VEL
LIN {X 0,Y 305.174,Z 831.81,A -85,B 0,C 180,E1 13988.433,E2 13988.433} C_VEL
LIN {X 0,Y 304.852,Z 831.81,A -85,B 0,C 180,E1 14001.513,E2 14001.513} C_VEL
LIN {X 0,Y 305.212,Z 831.81,A -85,B 0,C 180,E1 14011.808,E2 14011.808} C_VEL
LIN {X 0,Y 306.045,Z 831.81,A -85,B 0,C 180,E1 14024.17,E2 14024.17} C_VEL
LIN {X 0,Y 306.842,Z 831.81,A -85,B 0,C 180,E1 14035.743,E2 14035.743} C_VEL
LIN {X 0,Y 306.852,Z 831.81,A -85,B 0,C 180,E1 14044.252,E2 14044.252} C_VEL
LIN {X 0,Y 306.123,Z 831.81,A -85,B 0,C 180,E1 14055.82,E2 14055.82} C_VEL
LIN {X 0,Y 305.299,Z 831.81,A -85,B 0,C 180,E1 14068.177,E2 14068.177} C_VEL
LIN {X 0,Y 304.808,Z 831.81,A -85,B 0,C 180,E1 14079.493,E2 14079.493} C_VEL
LIN {X 0,Y 304.814,Z 831.81,A -85,B 0,C 180,E1 14091.514,E2 14091.514} C_VEL
LIN {X 0,Y 305.18,Z 831.81,A -85,B 0,C 180,E1 14101.809,E2 14101.809} C_VEL
LIN {X 0,Y 305.784,Z 831.81,A -85,B 0,C 180,E1 14114.159,E2 14114.159} C_VEL
LIN {X 0,Y 306.757,Z 833.587,A -85,B 0,C 180,E1 14122.895,E2 14122.895} C_VEL
LIN {X 0,Y 318.729,Z 873.726,A -85,B 0,C 180,E1 14126.377,E2 14126.377} C_VEL
LIN {X 0,Y 320.129,Z 901.134,A -85,B 0,C 180,E1 14129.677,E2 14129.677} C_VEL
LIN {X 0,Y 314.311,Z 934.248,A -85,B 0,C 180,E1 14135.888,E2 14135.888} C_VEL
LIN {X 0,Y 310.765,Z 953.659,A -85,B 0,C 180,E1 14143.412,E2 14143.412} C_VEL
LIN {X 0,Y 310.02,Z 959.825,A -85,B 0,C 180,E1 14151.538,E2 14151.538} C_VEL
LIN {X 0,Y 312.848,Z 952.244,A -85,B 0,C 180,E1 14160.009,E2 14160.009} C_VEL
LIN {X 0,Y 319.262,Z 930.146,A -85,B 0,C 180,E1 14167.627,E2 14167.627} C_VEL
LIN {X 0,Y 327.1,Z 896.346,A -85,B 0,C 180,E1 14173.244,E2 14173.244} C_VEL
LIN {X 0,Y 317.582,Z 858.785,A -85,B 0,C 180,E1 14178.47,E2 14178.47} C_VEL
LIN {X 0,Y 304.961,Z 831.81,A -85,B 0,C 180,E1 14182.094,E2 14182.094} C_VEL
LIN {X 0,Y 305.294,Z 831.81,A -85,B 0,C 180,E1 14195.008,E2 14195.008} C_VEL
LIN {X 0,Y 306.04,Z 831.81,A -85,B 0,C 180,E1 14207.109,E2 14207.109} C_VEL
LIN {X 0,Y 307.323,Z 831.81,A -85,B 0,C 180,E1 14218.588,E2 14218.588} C_VEL
LIN {X 0,Y 306.526,Z 831.81,A -85,B 0,C 180,E1 14229.982,E2 14229.982} C_VEL
LIN {X 0,Y 305.646,Z 831.81,A -85,B 0,C 180,E1 14241.867,E2 14241.867} C_VEL
LIN {X 0,Y 305.065,Z 831.81,A -85,B 0,C 180,E1 14254.9,E2 14254.9} C_VEL
LIN {X 0,Y 305.13,Z 833.503,A -85,B 0,C 180,E1 14267.762,E2 14267.762} C_VEL
LIN {X 0,Y 330.782,Z 886.767,A -85,B 0,C 180,E1 14273.138,E2 14273.138} C_VEL
LIN {X 0,Y 333.643,Z 907.554,A -85,B 0,C 180,E1 14274.541,E2 14274.541} C_VEL
LIN {X 0,Y 325.317,Z 957.4,A -85,B 0,C 180,E1 14278.346,E2 14278.346} C_VEL
LIN {X 0,Y 315.864,Z 1000.109,A -85,B 0,C 180,E1 14284.762,E2 14284.762} C_VEL
LIN {X 0,Y 309.812,Z 1031.894,A -85,B 0,C 180,E1 14293.44,E2 14293.44} C_VEL
LIN {X 0,Y 308.79,Z 1049.337,A -85,B 0,C 180,E1 14302.943,E2 14302.943} C_VEL
LIN {X 0,Y 309.226,Z 1052.592,A -85,B 0,C 180,E1 14311.407,E2 14311.407} C_VEL
LIN {X 0,Y 308.818,Z 1042.909,A -85,B 0,C 180,E1 14320.496,E2 14320.496} C_VEL
LIN {X 0,Y 310.929,Z 1018.162,A -85,B 0,C 180,E1 14329.606,E2 14329.606} C_VEL
LIN {X 0,Y 317.503,Z 981.014,A -85,B 0,C 180,E1 14337.005,E2 14337.005} C_VEL
LIN {X 0,Y 325.166,Z 933.467,A -85,B 0,C 180,E1 14342.163,E2 14342.163} C_VEL
LIN {X 0,Y 327.507,Z 893.365,A -85,B 0,C 180,E1 14344.491,E2 14344.491} C_VEL
LIN {X 0,Y 314.383,Z 855.526,A -85,B 0,C 180,E1 14346.689,E2 14346.689} C_VEL
LIN {X 0,Y 299.716,Z 839.305,A -85,B 0,C 180,E1 14348.535,E2 14348.535} C_VEL
LIN {X 0,Y 297.103,Z 831.81,A -85,B 0,C 180,E1 14349.28,E2 14349.28} C_VEL
LIN {X 0,Y 296.801,Z 831.81,A -85,B 0,C 180,E1 14362.422,E2 14362.422} C_VEL
LIN {X 0,Y 297.273,Z 831.81,A -85,B 0,C 180,E1 14374.279,E2 14374.279} C_VEL
LIN {X 0,Y 298.193,Z 831.81,A -85,B 0,C 180,E1 14386.757,E2 14386.757} C_VEL
LIN {X 0,Y 298.995,Z 831.81,A -85,B 0,C 180,E1 14398.543,E2 14398.543} C_VEL
LIN {X 0,Y 298.482,Z 831.81,A -85,B 0,C 180,E1 14410.248,E2 14410.248} C_VEL
LIN {X 0,Y 297.658,Z 831.81,A -85,B 0,C 180,E1 14422.479,E2 14422.479} C_VEL
LIN {X 0,Y 297.016,Z 831.81,A -85,B 0,C 180,E1 14432.538,E2 14432.538} C_VEL
LIN {X 0,Y 296.768,Z 831.81,A -85,B 0,C 180,E1 14443.656,E2 14443.656} C_VEL
LIN {X 0,Y 296.81,Z 831.81,A -85,B 0,C 180,E1 14453.986,E2 14453.986} C_VEL
LIN {X 0,Y 297.191,Z 831.81,A -85,B 0,C 180,E1 14464.276,E2 14464.276} C_VEL
LIN {X 0,Y 297.969,Z 831.81,A -85,B 0,C 180,E1 14476.751,E2 14476.751} C_VEL
LIN {X 0,Y 298.516,Z 832.772,A -85,B 0,C 180,E1 14482.031,E2 14482.031} C_VEL
LIN {X 0,Y 311.075,Z 873.578,A -85,B 0,C 180,E1 14485.677,E2 14485.677} C_VEL
LIN {X 0,Y 312.734,Z 901.581,A -85,B 0,C 180,E1 14489.114,E2 14489.114} C_VEL
LIN {X 0,Y 306.761,Z 934.366,A -85,B 0,C 180,E1 14495.309,E2 14495.309} C_VEL
LIN {X 0,Y 302.951,Z 954.362,A -85,B 0,C 180,E1 14503.027,E2 14503.027} C_VEL
LIN {X 0,Y 302.211,Z 961.019,A -85,B 0,C 180,E1 14512.123,E2 14512.123} C_VEL
LIN {X 0,Y 305.491,Z 952.718,A -85,B 0,C 180,E1 14520.822,E2 14520.822} C_VEL
LIN {X 0,Y 312.382,Z 930.301,A -85,B 0,C 180,E1 14528.462,E2 14528.462} C_VEL
LIN {X 0,Y 319.914,Z 895.889,A -85,B 0,C 180,E1 14534.249,E2 14534.249} C_VEL
LIN {X 0,Y 309.484,Z 857.568,A -85,B 0,C 180,E1 14539.812,E2 14539.812} C_VEL
LIN {X 0,Y 296.973,Z 831.81,A -85,B 0,C 180,E1 14543.633,E2 14543.633} C_VEL
LIN {X 0,Y 297.179,Z 831.81,A -85,B 0,C 180,E1 14554.277,E2 14554.277} C_VEL
LIN {X 0,Y 297.984,Z 831.81,A -85,B 0,C 180,E1 14566.754,E2 14566.754} C_VEL
LIN {X 0,Y 299.299,Z 831.81,A -85,B 0,C 180,E1 14578.55,E2 14578.55} C_VEL
LIN {X 0,Y 298.471,Z 831.81,A -85,B 0,C 180,E1 14590.254,E2 14590.254} C_VEL
LIN {X 0,Y 297.602,Z 831.81,A -85,B 0,C 180,E1 14602.49,E2 14602.49} C_VEL
LIN {X 0,Y 297.053,Z 831.81,A -85,B 0,C 180,E1 14612.55,E2 14612.55} C_VEL
LIN {X 0,Y 296.885,Z 831.81,A -85,B 0,C 180,E1 14626.019,E2 14626.019} C_VEL
LIN {X 0,Y 323.266,Z 886.349,A -85,B 0,C 180,E1 14632.157,E2 14632.157} C_VEL
LIN {X 0,Y 326.923,Z 908.315,A -85,B 0,C 180,E1 14633.799,E2 14633.799} C_VEL
LIN {X 0,Y 318.092,Z 957.98,A -85,B 0,C 180,E1 14637.743,E2 14637.743} C_VEL
LIN {X 0,Y 308.047,Z 1000.762,A -85,B 0,C 180,E1 14644.466,E2 14644.466} C_VEL
LIN {X 0,Y 301.788,Z 1032.015,A -85,B 0,C 180,E1 14653.466,E2 14653.466} C_VEL
LIN {X 0,Y 300.821,Z 1048.176,A -85,B 0,C 180,E1 14662.755,E2 14662.755} C_VEL
LIN {X 0,Y 301.305,Z 1051.358,A -85,B 0,C 180,E1 14671.444,E2 14671.444} C_VEL
LIN {X 0,Y 300.848,Z 1041.424,A -85,B 0,C 180,E1 14680.83,E2 14680.83} C_VEL
LIN {X 0,Y 303.229,Z 1016.427,A -85,B 0,C 180,E1 14690.125,E2 14690.125} C_VEL
LIN {X 0,Y 310.148,Z 978.686,A -85,B 0,C 180,E1 14697.7,E2 14697.7} C_VEL
LIN {X 0,Y 318.088,Z 931.061,A -85,B 0,C 180,E1 14702.867,E2 14702.867} C_VEL
LIN {X 0,Y 320.225,Z 895.195,A -85,B 0,C 180,E1 14705.01,E2 14705.01} C_VEL
LIN {X 0,Y 299.716,Z 839.305,A -85,B 0,C 180,E1 14708.535,E2 14708.535} C_VEL
LIN {X 0,Y 292.203,Z 831.973,A -85,B 0,C 180,E1 14711.032,E2 14711.032} C_VEL
LIN {X 0,Y 288.773,Z 831.81,A -85,B 0,C 180,E1 14714.706,E2 14714.706} C_VEL
LIN {X 0,Y 288.854,Z 831.81,A -85,B 0,C 180,E1 14726.515,E2 14726.515} C_VEL
LIN {X 0,Y 289.643,Z 831.81,A -85,B 0,C 180,E1 14740.085,E2 14740.085} C_VEL
LIN {X 0,Y 290.669,Z 831.81,A -85,B 0,C 180,E1 14752.497,E2 14752.497} C_VEL
LIN {X 0,Y 290.8,Z 831.81,A -85,B 0,C 180,E1 14764.487,E2 14764.487} C_VEL
LIN {X 0,Y 289.949,Z 831.81,A -85,B 0,C 180,E1 14776.728,E2 14776.728} C_VEL
LIN {X 0,Y 289.068,Z 831.81,A -85,B 0,C 180,E1 14789.978,E2 14789.978} C_VEL
LIN {X 0,Y 288.722,Z 831.81,A -85,B 0,C 180,E1 14801.071,E2 14801.071} C_VEL
LIN {X 0,Y 288.761,Z 831.81,A -85,B 0,C 180,E1 14814.545,E2 14814.545} C_VEL
LIN {X 0,Y 289.215,Z 831.81,A -85,B 0,C 180,E1 14826.825,E2 14826.825} C_VEL
LIN {X 0,Y 290.188,Z 831.81,A -85,B 0,C 180,E1 14839.453,E2 14839.453} C_VEL
LIN {X 0,Y 290.458,Z 832.758,A -85,B 0,C 180,E1 14841.171,E2 14841.171} C_VEL
LIN {X 0,Y 303.523,Z 873.662,A -85,B 0,C 180,E1 14844.969,E2 14844.969} C_VEL
LIN {X 0,Y 305.119,Z 903.813,A -85,B 0,C 180,E1 14848.786,E2 14848.786} C_VEL
LIN {X 0,Y 298.863,Z 936.491,A -85,B 0,C 180,E1 14855.258,E2 14855.258} C_VEL
LIN {X 0,Y 294.918,Z 956.275,A -85,B 0,C 180,E1 14863.388,E2 14863.388} C_VEL
LIN {X 0,Y 294.429,Z 962.143,A -85,B 0,C 180,E1 14872.74,E2 14872.74} C_VEL
LIN {X 0,Y 298.245,Z 953.022,A -85,B 0,C 180,E1 14881.714,E2 14881.714} C_VEL
LIN {X 0,Y 305.834,Z 929.409,A -85,B 0,C 180,E1 14889.56,E2 14889.56} C_VEL
LIN {X 0,Y 312.737,Z 895.692,A -85,B 0,C 180,E1 14895.283,E2 14895.283} C_VEL
LIN {X 0,Y 301.909,Z 857.801,A -85,B 0,C 180,E1 14901.075,E2 14901.075} C_VEL
LIN {X 0,Y 288.852,Z 831.81,A -85,B 0,C 180,E1 14905.1,E2 14905.1} C_VEL
LIN {X 0,Y 289.21,Z 831.81,A -85,B 0,C 180,E1 14916.827,E2 14916.827} C_VEL
LIN {X 0,Y 290.233,Z 831.81,A -85,B 0,C 180,E1 14929.458,E2 14929.458} C_VEL
LIN {X 0,Y 290.987,Z 831.81,A -85,B 0,C 180,E1 14941.497,E2 14941.497} C_VEL
LIN {X 0,Y 290.023,Z 831.81,A -85,B 0,C 180,E1 14954.534,E2 14954.534} C_VEL
LIN {X 0,Y 289.285,Z 831.81,A -85,B 0,C 180,E1 14966.486,E2 14966.486} C_VEL
LIN {X 0,Y 288.854,Z 831.81,A -85,B 0,C 180,E1 14980.38,E2 14980.38} C_VEL
LIN {X 0,Y 288.893,Z 833.048,A -85,B 0,C 180,E1 14984.696,E2 14984.696} C_VEL
LIN {X 0,Y 315.469,Z 885.025,A -85,B 0,C 180,E1 14991.012,E2 14991.012} C_VEL
LIN {X 0,Y 320.26,Z 908.864,A -85,B 0,C 180,E1 14993.023,E2 14993.023} C_VEL
LIN {X 0,Y 310.915,Z 958.545,A -85,B 0,C 180,E1 14997.113,E2 14997.113} C_VEL
LIN {X 0,Y 300.673,Z 999.815,A -85,B 0,C 180,E1 15003.793,E2 15003.793} C_VEL
LIN {X 0,Y 294.028,Z 1030.712,A -85,B 0,C 180,E1 15012.919,E2 15012.919} C_VEL
LIN {X 0,Y 292.87,Z 1047.032,A -85,B 0,C 180,E1 15022.558,E2 15022.558} C_VEL
LIN {X 0,Y 293.396,Z 1050.123,A -85,B 0,C 180,E1 15031.482,E2 15031.482} C_VEL
LIN {X 0,Y 292.947,Z 1041.145,A -85,B 0,C 180,E1 15040.447,E2 15040.447} C_VEL
LIN {X 0,Y 295.051,Z 1017.298,A -85,B 0,C 180,E1 15049.923,E2 15049.923} C_VEL
LIN {X 0,Y 302.207,Z 979.949,A -85,B 0,C 180,E1 15057.881,E2 15057.881} C_VEL
LIN {X 0,Y 310.381,Z 933.076,A -85,B 0,C 180,E1 15063.266,E2 15063.266} C_VEL
LIN {X 0,Y 312.665,Z 896.212,A -85,B 0,C 180,E1 15065.603,E2 15065.603} C_VEL
LIN {X 0,Y 288.974,Z 831.81,A -85,B 0,C 180,E1 15070.072,E2 15070.072} C_VEL
LIN {X 0,Y 288.773,Z 831.81,A -85,B 0,C 180,E1 15074.706,E2 15074.706} C_VEL
LIN {X 0,Y 280.698,Z 831.81,A -85,B 0,C 180,E1 15081.647,E2 15081.647} C_VEL
LIN {X 0,Y 281.11,Z 831.81,A -85,B 0,C 180,E1 15092.967,E2 15092.967} C_VEL
LIN {X 0,Y 282.061,Z 831.81,A -85,B 0,C 180,E1 15105.985,E2 15105.985} C_VEL
LIN {X 0,Y 282.979,Z 831.81,A -85,B 0,C 180,E1 15118.46,E2 15118.46} C_VEL
LIN {X 0,Y 282.37,Z 831.81,A -85,B 0,C 180,E1 15130.839,E2 15130.839} C_VEL
LIN {X 0,Y 281.414,Z 831.81,A -85,B 0,C 180,E1 15143.854,E2 15143.854} C_VEL
LIN {X 0,Y 280.792,Z 831.81,A -85,B 0,C 180,E1 15154.573,E2 15154.573} C_VEL
LIN {X 0,Y 280.562,Z 831.81,A -85,B 0,C 180,E1 15167.459,E2 15167.459} C_VEL
LIN {X 0,Y 280.861,Z 831.81,A -85,B 0,C 180,E1 15179.115,E2 15179.115} C_VEL
LIN {X 0,Y 281.539,Z 831.81,A -85,B 0,C 180,E1 15192.754,E2 15192.754} C_VEL
LIN {X 0,Y 282.415,Z 833.293,A -85,B 0,C 180,E1 15200.279,E2 15200.279} C_VEL
LIN {X 0,Y 296.225,Z 875.24,A -85,B 0,C 180,E1 15204.391,E2 15204.391} C_VEL
LIN {X 0,Y 297.758,Z 904.193,A -85,B 0,C 180,E1 15208.174,E2 15208.174} C_VEL
LIN {X 0,Y 291.397,Z 936.028,A -85,B 0,C 180,E1 15214.48,E2 15214.48} C_VEL
LIN {X 0,Y 287.164,Z 956.83,A -85,B 0,C 180,E1 15222.9,E2 15222.9} C_VEL
LIN {X 0,Y 286.397,Z 963.447,A -85,B 0,C 180,E1 15231.985,E2 15231.985} C_VEL
LIN {X 0,Y 289.638,Z 956.761,A -85,B 0,C 180,E1 15240.718,E2 15240.718} C_VEL
LIN {X 0,Y 297.001,Z 936.02,A -85,B 0,C 180,E1 15248.899,E2 15248.899} C_VEL
LIN {X 0,Y 306.276,Z 902.968,A -85,B 0,C 180,E1 15255.106,E2 15255.106} C_VEL
LIN {X 0,Y 297.94,Z 866.529,A -85,B 0,C 180,E1 15261.07,E2 15261.07} C_VEL
LIN {X 0,Y 280.825,Z 831.81,A -85,B 0,C 180,E1 15266.886,E2 15266.886} C_VEL
LIN {X 0,Y 281.401,Z 831.81,A -85,B 0,C 180,E1 15280.688,E2 15280.688} C_VEL
LIN {X 0,Y 282.501,Z 831.81,A -85,B 0,C 180,E1 15293.602,E2 15293.602} C_VEL
LIN {X 0,Y 282.768,Z 831.81,A -85,B 0,C 180,E1 15304.621,E2 15304.621} C_VEL
LIN {X 0,Y 281.813,Z 831.81,A -85,B 0,C 180,E1 15317.232,E2 15317.232} C_VEL
LIN {X 0,Y 280.96,Z 831.81,A -85,B 0,C 180,E1 15330.877,E2 15330.877} C_VEL
LIN {X 0,Y 281.009,Z 833.648,A -85,B 0,C 180,E1 15343.006,E2 15343.006} C_VEL
LIN {X 0,Y 307.282,Z 882.717,A -85,B 0,C 180,E1 15349.684,E2 15349.684} C_VEL
LIN {X 0,Y 313.686,Z 909.616,A -85,B 0,C 180,E1 15352.218,E2 15352.218} C_VEL
LIN {X 0,Y 303.765,Z 959.108,A -85,B 0,C 180,E1 15356.451,E2 15356.451} C_VEL
LIN {X 0,Y 292.899,Z 1000.544,A -85,B 0,C 180,E1 15363.458,E2 15363.458} C_VEL
LIN {X 0,Y 285.952,Z 1031.05,A -85,B 0,C 180,E1 15373.03,E2 15373.03} C_VEL
LIN {X 0,Y 284.901,Z 1045.884,A -85,B 0,C 180,E1 15382.348,E2 15382.348} C_VEL
LIN {X 0,Y 285.472,Z 1048.882,A -85,B 0,C 180,E1 15391.524,E2 15391.524} C_VEL
LIN {X 0,Y 284.954,Z 1039.717,A -85,B 0,C 180,E1 15400.743,E2 15400.743} C_VEL
LIN {X 0,Y 287.384,Z 1015.587,A -85,B 0,C 180,E1 15410.478,E2 15410.478} C_VEL
LIN {X 0,Y 294.682,Z 978.803,A -85,B 0,C 180,E1 15418.448,E2 15418.448} C_VEL
LIN {X 0,Y 303.273,Z 931.236,A -85,B 0,C 180,E1 15423.968,E2 15423.968} C_VEL
LIN {X 0,Y 305.381,Z 898.008,A -85,B 0,C 180,E1 15426.161,E2 15426.161} C_VEL
LIN {X 0,Y 280.92,Z 831.81,A -85,B 0,C 180,E1 15430.937,E2 15430.937} C_VEL
LIN {X 0,Y 280.698,Z 831.81,A -85,B 0,C 180,E1 15441.647,E2 15441.647} C_VEL
LIN {X 0,Y 272.827,Z 831.81,A -85,B 0,C 180,E1 15448.8,E2 15448.8} C_VEL
LIN {X 0,Y 273.717,Z 831.81,A -85,B 0,C 180,E1 15462.242,E2 15462.242} C_VEL
LIN {X 0,Y 274.762,Z 831.81,A -85,B 0,C 180,E1 15475.244,E2 15475.244} C_VEL
LIN {X 0,Y 274.761,Z 831.81,A -85,B 0,C 180,E1 15484.749,E2 15484.749} C_VEL
LIN {X 0,Y 273.814,Z 831.81,A -85,B 0,C 180,E1 15497.745,E2 15497.745} C_VEL
LIN {X 0,Y 272.913,Z 831.81,A -85,B 0,C 180,E1 15510.471,E2 15510.471} C_VEL
LIN {X 0,Y 272.461,Z 831.81,A -85,B 0,C 180,E1 15524.123,E2 15524.123} C_VEL
LIN {X 0,Y 272.809,Z 831.81,A -85,B 0,C 180,E1 15538.099,E2 15538.099} C_VEL
LIN {X 0,Y 273.463,Z 831.81,A -85,B 0,C 180,E1 15552.228,E2 15552.228} C_VEL
LIN {X 0,Y 274.257,Z 833.209,A -85,B 0,C 180,E1 15559.293,E2 15559.293} C_VEL
LIN {X 0,Y 288.864,Z 876.259,A -85,B 0,C 180,E1 15563.724,E2 15563.724} C_VEL
LIN {X 0,Y 290.044,Z 907.094,A -85,B 0,C 180,E1 15567.904,E2 15567.904} C_VEL
LIN {X 0,Y 283.414,Z 938.843,A -85,B 0,C 180,E1 15574.606,E2 15574.606} C_VEL
LIN {X 0,Y 279.078,Z 958.92,A -85,B 0,C 180,E1 15583.425,E2 15583.425} C_VEL
LIN {X 0,Y 278.315,Z 964.543,A -85,B 0,C 180,E1 15590.757,E2 15590.757} C_VEL
LIN {X 0,Y 281.777,Z 958.571,A -85,B 0,C 180,E1 15600.772,E2 15600.772} C_VEL
LIN {X 0,Y 289.702,Z 937.768,A -85,B 0,C 180,E1 15609.43,E2 15609.43} C_VEL
LIN {X 0,Y 299.357,Z 904.014,A -85,B 0,C 180,E1 15615.996,E2 15615.996} C_VEL
LIN {X 0,Y 291.032,Z 867.995,A -85,B 0,C 180,E1 15622.217,E2 15622.217} C_VEL
LIN {X 0,Y 272.835,Z 831.81,A -85,B 0,C 180,E1 15628.9,E2 15628.9} C_VEL
LIN {X 0,Y 273.483,Z 831.81,A -85,B 0,C 180,E1 15642.233,E2 15642.233} C_VEL
LIN {X 0,Y 274.703,Z 831.81,A -85,B 0,C 180,E1 15655.25,E2 15655.25} C_VEL
LIN {X 0,Y 274.595,Z 831.81,A -85,B 0,C 180,E1 15667.945,E2 15667.945} C_VEL
LIN {X 0,Y 273.48,Z 831.81,A -85,B 0,C 180,E1 15681.147,E2 15681.147} C_VEL
LIN {X 0,Y 272.894,Z 831.81,A -85,B 0,C 180,E1 15691.896,E2 15691.896} C_VEL
LIN {X 0,Y 272.821,Z 833.566,A -85,B 0,C 180,E1 15701.052,E2 15701.052} C_VEL
LIN {X 0,Y 298.969,Z 880.317,A -85,B 0,C 180,E1 15708.212,E2 15708.212} C_VEL
LIN {X 0,Y 307.171,Z 910.425,A -85,B 0,C 180,E1 15711.379,E2 15711.379} C_VEL
LIN {X 0,Y 297.026,Z 958.372,A -85,B 0,C 180,E1 15715.585,E2 15715.585} C_VEL
LIN {X 0,Y 285.595,Z 999.611,A -85,B 0,C 180,E1 15722.723,E2 15722.723} C_VEL
LIN {X 0,Y 278.142,Z 1030.003,A -85,B 0,C 180,E1 15732.538,E2 15732.538} C_VEL
LIN {X 0,Y 276.958,Z 1044.738,A -85,B 0,C 180,E1 15742.127,E2 15742.127} C_VEL
LIN {X 0,Y 277.559,Z 1047.642,A -85,B 0,C 180,E1 15751.567,E2 15751.567} C_VEL
LIN {X 0,Y 276.968,Z 1038.289,A -85,B 0,C 180,E1 15761.057,E2 15761.057} C_VEL
LIN {X 0,Y 279.444,Z 1015.127,A -85,B 0,C 180,E1 15770.671,E2 15770.671} C_VEL
LIN {X 0,Y 287.025,Z 978.422,A -85,B 0,C 180,E1 15778.902,E2 15778.902} C_VEL
LIN {X 0,Y 295.865,Z 931.517,A -85,B 0,C 180,E1 15784.537,E2 15784.537} C_VEL
LIN {X 0,Y 298.186,Z 900.005,A -85,B 0,C 180,E1 15786.72,E2 15786.72} C_VEL
LIN {X 0,Y 272.764,Z 831.81,A -85,B 0,C 180,E1 15792.063,E2 15792.063} C_VEL
LIN {X 0,Y 272.627,Z 831.81,A -85,B 0,C 180,E1 15804.228,E2 15804.228} C_VEL
LIN {X 0,Y 272.827,Z 831.81,A -85,B 0,C 180,E1 15808.8,E2 15808.8} C_VEL
LIN {X 0,Y 265.036,Z 831.81,A -85,B 0,C 180,E1 15816.216,E2 15816.216} C_VEL
LIN {X 0,Y 266.201,Z 831.81,A -85,B 0,C 180,E1 15828.487,E2 15828.487} C_VEL
LIN {X 0,Y 267.231,Z 831.81,A -85,B 0,C 180,E1 15841.624,E2 15841.624} C_VEL
LIN {X 0,Y 265.985,Z 831.81,A -85,B 0,C 180,E1 15854.874,E2 15854.874} C_VEL
LIN {X 0,Y 265.016,Z 831.81,A -85,B 0,C 180,E1 15867.43,E2 15867.43} C_VEL
LIN {X 0,Y 264.481,Z 831.81,A -85,B 0,C 180,E1 15881.287,E2 15881.287} C_VEL
LIN {X 0,Y 264.47,Z 831.81,A -85,B 0,C 180,E1 15892.95,E2 15892.95} C_VEL
LIN {X 0,Y 264.933,Z 831.81,A -85,B 0,C 180,E1 15904.557,E2 15904.557} C_VEL
LIN {X 0,Y 265.946,Z 832.313,A -85,B 0,C 180,E1 15918.198,E2 15918.198} C_VEL
LIN {X 0,Y 281.243,Z 875.331,A -85,B 0,C 180,E1 15922.801,E2 15922.801} C_VEL
LIN {X 0,Y 282.664,Z 907.899,A -85,B 0,C 180,E1 15927.307,E2 15927.307} C_VEL
LIN {X 0,Y 275.641,Z 940.273,A -85,B 0,C 180,E1 15934.341,E2 15934.341} C_VEL
LIN {X 0,Y 271.236,Z 959.904,A -85,B 0,C 180,E1 15943.19,E2 15943.19} C_VEL
LIN {X 0,Y 270.604,Z 965.872,A -85,B 0,C 180,E1 15952.284,E2 15952.284} C_VEL
LIN {X 0,Y 274.476,Z 959.155,A -85,B 0,C 180,E1 15961.684,E2 15961.684} C_VEL
LIN {X 0,Y 283.124,Z 937.525,A -85,B 0,C 180,E1 15970.533,E2 15970.533} C_VEL
LIN {X 0,Y 292.432,Z 903.735,A -85,B 0,C 180,E1 15977.182,E2 15977.182} C_VEL
LIN {X 0,Y 284.013,Z 868.94,A -85,B 0,C 180,E1 15983.529,E2 15983.529} C_VEL
LIN {X 0,Y 264.825,Z 831.81,A -85,B 0,C 180,E1 15990.853,E2 15990.853} C_VEL
LIN {X 0,Y 265.665,Z 831.81,A -85,B 0,C 180,E1 16005.107,E2 16005.107} C_VEL
LIN {X 0,Y 267.214,Z 831.81,A -85,B 0,C 180,E1 16018.376,E2 16018.376} C_VEL
LIN {X 0,Y 266.231,Z 831.81,A -85,B 0,C 180,E1 16031.512,E2 16031.512} C_VEL
LIN {X 0,Y 265.099,Z 831.81,A -85,B 0,C 180,E1 16045.43,E2 16045.43} C_VEL
LIN {X 0,Y 264.675,Z 833.354,A -85,B 0,C 180,E1 16058.849,E2 16058.849} C_VEL
LIN {X 0,Y 290.839,Z 878.41,A -85,B 0,C 180,E1 16066.663,E2 16066.663} C_VEL
LIN {X 0,Y 300.665,Z 911.633,A -85,B 0,C 180,E1 16070.527,E2 16070.527} C_VEL
LIN {X 0,Y 289.651,Z 960.442,A -85,B 0,C 180,E1 16075.038,E2 16075.038} C_VEL
LIN {X 0,Y 277.836,Z 1000.291,A -85,B 0,C 180,E1 16082.338,E2 16082.338} C_VEL
LIN {X 0,Y 270.094,Z 1030.095,A -85,B 0,C 180,E1 16092.578,E2 16092.578} C_VEL
LIN {X 0,Y 269.146,Z 1044.895,A -85,B 0,C 180,E1 16103.526,E2 16103.526} C_VEL
LIN {X 0,Y 269.631,Z 1046.399,A -85,B 0,C 180,E1 16111.613,E2 16111.613} C_VEL
LIN {X 0,Y 268.981,Z 1036.849,A -85,B 0,C 180,E1 16121.389,E2 16121.389} C_VEL
LIN {X 0,Y 271.908,Z 1012.323,A -85,B 0,C 180,E1 16131.603,E2 16131.603} C_VEL
LIN {X 0,Y 280.001,Z 975.181,A -85,B 0,C 180,E1 16139.861,E2 16139.861} C_VEL
LIN {X 0,Y 289.172,Z 927.711,A -85,B 0,C 180,E1 16145.462,E2 16145.462} C_VEL
LIN {X 0,Y 290.679,Z 901.078,A -85,B 0,C 180,E1 16147.378,E2 16147.378} C_VEL
LIN {X 0,Y 265.874,Z 835.945,A -85,B 0,C 180,E1 16152.595,E2 16152.595} C_VEL
LIN {X 0,Y 264.64,Z 831.81,A -85,B 0,C 180,E1 16153.261,E2 16153.261} C_VEL
LIN {X 0,Y 264.646,Z 831.81,A -85,B 0,C 180,E1 16166.986,E2 16166.986} C_VEL
LIN {X 0,Y 265.036,Z 831.81,A -85,B 0,C 180,E1 16176.216,E2 16176.216} C_VEL
LIN {X 0,Y 257.666,Z 831.81,A -85,B 0,C 180,E1 16183.884,E2 16183.884} C_VEL
LIN {X 0,Y 258.747,Z 831.81,A -85,B 0,C 180,E1 16194.949,E2 16194.949} C_VEL
LIN {X 0,Y 258.731,Z 831.81,A -85,B 0,C 180,E1 16205.044,E2 16205.044} C_VEL
LIN {X 0,Y 257.63,Z 831.81,A -85,B 0,C 180,E1 16218.901,E2 16218.901} C_VEL
LIN {X 0,Y 256.671,Z 831.81,A -85,B 0,C 180,E1 16230.985,E2 16230.985} C_VEL
LIN {X 0,Y 256.401,Z 831.81,A -85,B 0,C 180,E1 16242.892,E2 16242.892} C_VEL
LIN {X 0,Y 256.522,Z 831.81,A -85,B 0,C 180,E1 16255.805,E2 16255.805} C_VEL
LIN {X 0,Y 257.004,Z 831.81,A -85,B 0,C 180,E1 16267.43,E2 16267.43} C_VEL
LIN {X 0,Y 258.107,Z 833.796,A -85,B 0,C 180,E1 16277.181,E2 16277.181} C_VEL
LIN {X 0,Y 273.78,Z 876.262,A -85,B 0,C 180,E1 16282.034,E2 16282.034} C_VEL
LIN {X 0,Y 275.371,Z 908.416,A -85,B 0,C 180,E1 16286.643,E2 16286.643} C_VEL
LIN {X 0,Y 267.876,Z 941.666,A -85,B 0,C 180,E1 16294.06,E2 16294.06} C_VEL
LIN {X 0,Y 263.264,Z 961.364,A -85,B 0,C 180,E1 16303.33,E2 16303.33} C_VEL
LIN {X 0,Y 262.67,Z 967.084,A -85,B 0,C 180,E1 16312.056,E2 16312.056} C_VEL
LIN {X 0,Y 266.444,Z 961.306,A -85,B 0,C 180,E1 16321.508,E2 16321.508} C_VEL
LIN {X 0,Y 275.304,Z 940.854,A -85,B 0,C 180,E1 16330.683,E2 16330.683} C_VEL
LIN {X 0,Y 285.783,Z 908.108,A -85,B 0,C 180,E1 16337.545,E2 16337.545} C_VEL
LIN {X 0,Y 278.026,Z 872.352,A -85,B 0,C 180,E1 16344.472,E2 16344.472} C_VEL
LIN {X 0,Y 258.89,Z 837.187,A -85,B 0,C 180,E1 16352.206,E2 16352.206} C_VEL
LIN {X 0,Y 256.858,Z 831.81,A -85,B 0,C 180,E1 16353.7,E2 16353.7} C_VEL
LIN {X 0,Y 257.943,Z 831.81,A -85,B 0,C 180,E1 16368.12,E2 16368.12} C_VEL
LIN {X 0,Y 259.203,Z 831.81,A -85,B 0,C 180,E1 16378.326,E2 16378.326} C_VEL
LIN {X 0,Y 258.145,Z 831.81,A -85,B 0,C 180,E1 16391.878,E2 16391.878} C_VEL
LIN {X 0,Y 257.102,Z 831.81,A -85,B 0,C 180,E1 16403.812,E2 16403.812} C_VEL
LIN {X 0,Y 256.808,Z 833.821,A -85,B 0,C 180,E1 16416.493,E2 16416.493} C_VEL
LIN {X 0,Y 282.073,Z 875.347,A -85,B 0,C 180,E1 16424.792,E2 16424.792} C_VEL
LIN {X 0,Y 294.258,Z 912.655,A -85,B 0,C 180,E1 16429.62,E2 16429.62} C_VEL
LIN {X 0,Y 282.848,Z 960.229,A -85,B 0,C 180,E1 16434.168,E2 16434.168} C_VEL
LIN {X 0,Y 270.102,Z 1000.931,A -85,B 0,C 180,E1 16441.931,E2 16441.931} C_VEL
LIN {X 0,Y 262.156,Z 1029.693,A -85,B 0,C 180,E1 16452.369,E2 16452.369} C_VEL
LIN {X 0,Y 261.169,Z 1043.739,A -85,B 0,C 180,E1 16463.327,E2 16463.327} C_VEL
LIN {X 0,Y 261.714,Z 1045.152,A -85,B 0,C 180,E1 16471.662,E2 16471.662} C_VEL
LIN {X 0,Y 261.027,Z 1035.375,A -85,B 0,C 180,E1 16481.741,E2 16481.741} C_VEL
LIN {X 0,Y 264.063,Z 1011.544,A -85,B 0,C 180,E1 16491.935,E2 16491.935} C_VEL
LIN {X 0,Y 272.448,Z 974.637,A -85,B 0,C 180,E1 16500.414,E2 16500.414} C_VEL
LIN {X 0,Y 281.887,Z 927.569,A -85,B 0,C 180,E1 16506.126,E2 16506.126} C_VEL
LIN {X 0,Y 283.187,Z 902.308,A -85,B 0,C 180,E1 16508.044,E2 16508.044} C_VEL
LIN {X 0,Y 260.267,Z 840.879,A -85,B 0,C 180,E1 16513.202,E2 16513.202} C_VEL
LIN {X 0,Y 256.592,Z 831.81,A -85,B 0,C 180,E1 16514.064,E2 16514.064} C_VEL
LIN {X 0,Y 256.546,Z 831.81,A -85,B 0,C 180,E1 16525.803,E2 16525.803} C_VEL
LIN {X 0,Y 257.182,Z 831.81,A -85,B 0,C 180,E1 16537.442,E2 16537.442} C_VEL
LIN {X 0,Y 257.666,Z 831.81,A -85,B 0,C 180,E1 16543.884,E2 16543.884} C_VEL
LIN {X 0,Y 250.381,Z 831.81,A -85,B 0,C 180,E1 16551.749,E2 16551.749} C_VEL
LIN {X 0,Y 250.85,Z 831.81,A -85,B 0,C 180,E1 16563.445,E2 16563.445} C_VEL
LIN {X 0,Y 249.785,Z 831.81,A -85,B 0,C 180,E1 16575.864,E2 16575.864} C_VEL
LIN {X 0,Y 248.796,Z 831.81,A -85,B 0,C 180,E1 16587.817,E2 16587.817} C_VEL
LIN {X 0,Y 248.278,Z 831.81,A -85,B 0,C 180,E1 16600.178,E2 16600.178} C_VEL
LIN {X 0,Y 248.489,Z 831.81,A -85,B 0,C 180,E1 16615.532,E2 16615.532} C_VEL
LIN {X 0,Y 249.206,Z 831.81,A -85,B 0,C 180,E1 16630.432,E2 16630.432} C_VEL
LIN {X 0,Y 249.826,Z 833.331,A -85,B 0,C 180,E1 16635.949,E2 16635.949} C_VEL
LIN {X 0,Y 265.895,Z 875.403,A -85,B 0,C 180,E1 16640.969,E2 16640.969} C_VEL
LIN {X 0,Y 268.034,Z 909.313,A -85,B 0,C 180,E1 16646.003,E2 16646.003} C_VEL
LIN {X 0,Y 260.395,Z 941.803,A -85,B 0,C 180,E1 16653.34,E2 16653.34} C_VEL
LIN {X 0,Y 255.468,Z 962.084,A -85,B 0,C 180,E1 16662.87,E2 16662.87} C_VEL
LIN {X 0,Y 254.889,Z 968.29,A -85,B 0,C 180,E1 16672.767,E2 16672.767} C_VEL
LIN {X 0,Y 259.261,Z 961.858,A -85,B 0,C 180,E1 16682.557,E2 16682.557} C_VEL
LIN {X 0,Y 268.74,Z 941.107,A -85,B 0,C 180,E1 16691.769,E2 16691.769} C_VEL
LIN {X 0,Y 279.035,Z 909.741,A -85,B 0,C 180,E1 16698.469,E2 16698.469} C_VEL
LIN {X 0,Y 271.796,Z 874.916,A -85,B 0,C 180,E1 16705.611,E2 16705.611} C_VEL
LIN {X 0,Y 252.552,Z 838.572,A -85,B 0,C 180,E1 16714.212,E2 16714.212} C_VEL
LIN {X 0,Y 248.928,Z 831.81,A -85,B 0,C 180,E1 16716.658,E2 16716.658} C_VEL
LIN {X 0,Y 250.237,Z 831.81,A -85,B 0,C 180,E1 16731.283,E2 16731.283} C_VEL
LIN {X 0,Y 250.758,Z 831.81,A -85,B 0,C 180,E1 16743.101,E2 16743.101} C_VEL
LIN {X 0,Y 249.725,Z 831.81,A -85,B 0,C 180,E1 16755.875,E2 16755.875} C_VEL
LIN {X 0,Y 248.785,Z 831.81,A -85,B 0,C 180,E1 16767.815,E2 16767.815} C_VEL
LIN {X 0,Y 248.733,Z 833.408,A -85,B 0,C 180,E1 16773.642,E2 16773.642} C_VEL
LIN {X 0,Y 274.118,Z 874.081,A -85,B 0,C 180,E1 16782.979,E2 16782.979} C_VEL
LIN {X 0,Y 287.853,Z 913.203,A -85,B 0,C 180,E1 16788.622,E2 16788.622} C_VEL
LIN {X 0,Y 276.05,Z 960.425,A -85,B 0,C 180,E1 16793.31,E2 16793.31} C_VEL
LIN {X 0,Y 262.901,Z 1000.051,A -85,B 0,C 180,E1 16801.091,E2 16801.091} C_VEL
LIN {X 0,Y 254.432,Z 1028.374,A -85,B 0,C 180,E1 16811.659,E2 16811.659} C_VEL
LIN {X 0,Y 253.084,Z 1041.584,A -85,B 0,C 180,E1 16821.686,E2 16821.686} C_VEL
LIN {X 0,Y 253.782,Z 1043.902,A -85,B 0,C 180,E1 16831.714,E2 16831.714} C_VEL
LIN {X 0,Y 253.092,Z 1033.879,A -85,B 0,C 180,E1 16842.115,E2 16842.115} C_VEL
LIN {X 0,Y 256.447,Z 1009.715,A -85,B 0,C 180,E1 16852.622,E2 16852.622} C_VEL
LIN {X 0,Y 265.257,Z 972.335,A -85,B 0,C 180,E1 16861.281,E2 16861.281} C_VEL
LIN {X 0,Y 274.891,Z 925.92,A -85,B 0,C 180,E1 16866.941,E2 16866.941} C_VEL
LIN {X 0,Y 275.817,Z 903.331,A -85,B 0,C 180,E1 16868.751,E2 16868.751} C_VEL
LIN {X 0,Y 254.108,Z 844.841,A -85,B 0,C 180,E1 16873.951,E2 16873.951} C_VEL
LIN {X 0,Y 248.446,Z 831.81,A -85,B 0,C 180,E1 16875.369,E2 16875.369} C_VEL
LIN {X 0,Y 248.601,Z 831.81,A -85,B 0,C 180,E1 16888.738,E2 16888.738} C_VEL
LIN {X 0,Y 249.411,Z 831.81,A -85,B 0,C 180,E1 16900.58,E2 16900.58} C_VEL
LIN {X 0,Y 250.381,Z 831.81,A -85,B 0,C 180,E1 16911.749,E2 16911.749} C_VEL
LIN {X 0,Y 242.931,Z 831.81,A -85,B 0,C 180,E1 16919.835,E2 16919.835} C_VEL
LIN {X 0,Y 241.885,Z 831.81,A -85,B 0,C 180,E1 16933.48,E2 16933.48} C_VEL
LIN {X 0,Y 240.74,Z 831.81,A -85,B 0,C 180,E1 16948.212,E2 16948.212} C_VEL
LIN {X 0,Y 240.11,Z 831.81,A -85,B 0,C 180,E1 16963.379,E2 16963.379} C_VEL
LIN {X 0,Y 240.529,Z 831.81,A -85,B 0,C 180,E1 16978.4,E2 16978.4} C_VEL
LIN {X 0,Y 241.365,Z 831.81,A -85,B 0,C 180,E1 16993.564,E2 16993.564} C_VEL
LIN {X 0,Y 241.919,Z 834.268,A -85,B 0,C 180,E1 16994.739,E2 16994.739} C_VEL
LIN {X 0,Y 258.028,Z 874.871,A -85,B 0,C 180,E1 16999.903,E2 16999.903} C_VEL
LIN {X 0,Y 260.744,Z 910.088,A -85,B 0,C 180,E1 17005.306,E2 17005.306} C_VEL
LIN {X 0,Y 252.706,Z 942.938,A -85,B 0,C 180,E1 17012.918,E2 17012.918} C_VEL
LIN {X 0,Y 247.674,Z 962.744,A -85,B 0,C 180,E1 17022.383,E2 17022.383} C_VEL
LIN {X 0,Y 247.157,Z 969.497,A -85,B 0,C 180,E1 17033.521,E2 17033.521} C_VEL
LIN {X 0,Y 252.202,Z 962.251,A -85,B 0,C 180,E1 17043.728,E2 17043.728} C_VEL
LIN {X 0,Y 262.45,Z 940.86,A -85,B 0,C 180,E1 17053.035,E2 17053.035} C_VEL
LIN {X 0,Y 272.269,Z 909.638,A -85,B 0,C 180,E1 17059.84,E2 17059.84} C_VEL
LIN {X 0,Y 265.182,Z 876.37,A -85,B 0,C 180,E1 17067.069,E2 17067.069} C_VEL
LIN {X 0,Y 247.878,Z 843.89,A -85,B 0,C 180,E1 17075.594,E2 17075.594} C_VEL
LIN {X 0,Y 241.073,Z 831.81,A -85,B 0,C 180,E1 17079.746,E2 17079.746} C_VEL
LIN {X 0,Y 242.578,Z 831.81,A -85,B 0,C 180,E1 17094.619,E2 17094.619} C_VEL
LIN {X 0,Y 242.674,Z 831.81,A -85,B 0,C 180,E1 17105.386,E2 17105.386} C_VEL
LIN {X 0,Y 241.625,Z 831.81,A -85,B 0,C 180,E1 17116.422,E2 17116.422} C_VEL
LIN {X 0,Y 240.845,Z 833.704,A -85,B 0,C 180,E1 17130.425,E2 17130.425} C_VEL
LIN {X 0,Y 264.404,Z 869.708,A -85,B 0,C 180,E1 17140.359,E2 17140.359} C_VEL
LIN {X 0,Y 279.931,Z 908.456,A -85,B 0,C 180,E1 17146.75,E2 17146.75} C_VEL
LIN {X 0,Y 279.565,Z 924.125,A -85,B 0,C 180,E1 17148.391,E2 17148.391} C_VEL
LIN {X 0,Y 266.001,Z 970.628,A -85,B 0,C 180,E1 17153.962,E2 17153.962} C_VEL
LIN {X 0,Y 252.635,Z 1007.633,A -85,B 0,C 180,E1 17162.741,E2 17162.741} C_VEL
LIN {X 0,Y 245.548,Z 1031.992,A -85,B 0,C 180,E1 17173.853,E2 17173.853} C_VEL
LIN {X 0,Y 245.448,Z 1042.347,A -85,B 0,C 180,E1 17184.679,E2 17184.679} C_VEL
LIN {X 0,Y 245.849,Z 1042.652,A -85,B 0,C 180,E1 17191.769,E2 17191.769} C_VEL
LIN {X 0,Y 245.167,Z 1032.382,A -85,B 0,C 180,E1 17202.513,E2 17202.513} C_VEL
LIN {X 0,Y 248.924,Z 1007.818,A -85,B 0,C 180,E1 17213.346,E2 17213.346} C_VEL
LIN {X 0,Y 258.131,Z 970.128,A -85,B 0,C 180,E1 17222.173,E2 17222.173} C_VEL
LIN {X 0,Y 268.268,Z 922.402,A -85,B 0,C 180,E1 17227.96,E2 17227.96} C_VEL
LIN {X 0,Y 268,Z 902.783,A -85,B 0,C 180,E1 17229.66,E2 17229.66} C_VEL
LIN {X 0,Y 246.525,Z 845.608,A -85,B 0,C 180,E1 17235.069,E2 17235.069} C_VEL
LIN {X 0,Y 240.279,Z 831.81,A -85,B 0,C 180,E1 17236.579,E2 17236.579} C_VEL
LIN {X 0,Y 240.662,Z 831.81,A -85,B 0,C 180,E1 17251.77,E2 17251.77} C_VEL
LIN {X 0,Y 241.848,Z 831.81,A -85,B 0,C 180,E1 17266.556,E2 17266.556} C_VEL
LIN {X 0,Y 242.931,Z 831.81,A -85,B 0,C 180,E1 17279.835,E2 17279.835} C_VEL
LIN {X 0,Y 234.266,Z 831.81,A -85,B 0,C 180,E1 17288.154,E2 17288.154} C_VEL
LIN {X 0,Y 233.209,Z 831.81,A -85,B 0,C 180,E1 17300.968,E2 17300.968} C_VEL
LIN {X 0,Y 232.174,Z 831.81,A -85,B 0,C 180,E1 17315.211,E2 17315.211} C_VEL
LIN {X 0,Y 232.069,Z 831.81,A -85,B 0,C 180,E1 17328.763,E2 17328.763} C_VEL
LIN {X 0,Y 232.622,Z 831.81,A -85,B 0,C 180,E1 17341.724,E2 17341.724} C_VEL
LIN {X 0,Y 233.411,Z 833.106,A -85,B 0,C 180,E1 17353.254,E2 17353.254} C_VEL
LIN {X 0,Y 250.495,Z 875.534,A -85,B 0,C 180,E1 17358.933,E2 17358.933} C_VEL
LIN {X 0,Y 253.873,Z 908.895,A -85,B 0,C 180,E1 17364.26,E2 17364.26} C_VEL
LIN {X 0,Y 245.512,Z 941.905,A -85,B 0,C 180,E1 17371.77,E2 17371.77} C_VEL
LIN {X 0,Y 240.035,Z 962.885,A -85,B 0,C 180,E1 17381.498,E2 17381.498} C_VEL
LIN {X 0,Y 239.136,Z 970.715,A -85,B 0,C 180,E1 17393.052,E2 17393.052} C_VEL
LIN {X 0,Y 244.578,Z 963.765,A -85,B 0,C 180,E1 17404.159,E2 17404.159} C_VEL
LIN {X 0,Y 255.333,Z 942.76,A -85,B 0,C 180,E1 17413.732,E2 17413.732} C_VEL
LIN {X 0,Y 265.721,Z 913.242,A -85,B 0,C 180,E1 17420.442,E2 17420.442} C_VEL
LIN {X 0,Y 259.301,Z 879.642,A -85,B 0,C 180,E1 17428.216,E2 17428.216} C_VEL
LIN {X 0,Y 242.234,Z 845.925,A -85,B 0,C 180,E1 17437.685,E2 17437.685} C_VEL
LIN {X 0,Y 233.39,Z 831.81,A -85,B 0,C 180,E1 17443.961,E2 17443.961} C_VEL
LIN {X 0,Y 235.125,Z 831.81,A -85,B 0,C 180,E1 17458.154,E2 17458.154} C_VEL
LIN {X 0,Y 234.265,Z 831.81,A -85,B 0,C 180,E1 17469.324,E2 17469.324} C_VEL
LIN {X 0,Y 233.158,Z 831.81,A -85,B 0,C 180,E1 17480.981,E2 17480.981} C_VEL
LIN {X 0,Y 232.904,Z 833.555,A -85,B 0,C 180,E1 17486.404,E2 17486.404} C_VEL
LIN {X 0,Y 252.636,Z 862.421,A -85,B 0,C 180,E1 17496.523,E2 17496.523} C_VEL
LIN {X 0,Y 270.735,Z 900.151,A -85,B 0,C 180,E1 17504.072,E2 17504.072} C_VEL
LIN {X 0,Y 274.272,Z 921.015,A -85,B 0,C 180,E1 17507.066,E2 17507.066} C_VEL
LIN {X 0,Y 260.285,Z 967.617,A -85,B 0,C 180,E1 17512.517,E2 17512.517} C_VEL
LIN {X 0,Y 245.918,Z 1005.468,A -85,B 0,C 180,E1 17521.43,E2 17521.43} C_VEL
LIN {X 0,Y 237.749,Z 1030.937,A -85,B 0,C 180,E1 17533.308,E2 17533.308} C_VEL
LIN {X 0,Y 237.484,Z 1041.175,A -85,B 0,C 180,E1 17544.5,E2 17544.5} C_VEL
LIN {X 0,Y 237.677,Z 1040.523,A -85,B 0,C 180,E1 17553.661,E2 17553.661} C_VEL
LIN {X 0,Y 237.598,Z 1027.825,A -85,B 0,C 180,E1 17564.803,E2 17564.803} C_VEL
LIN {X 0,Y 243.01,Z 999.963,A -85,B 0,C 180,E1 17575.936,E2 17575.936} C_VEL
LIN {X 0,Y 253.217,Z 959.661,A -85,B 0,C 180,E1 17584.444,E2 17584.444} C_VEL
LIN {X 0,Y 262.363,Z 911.328,A -85,B 0,C 180,E1 17589.636,E2 17589.636} C_VEL
LIN {X 0,Y 244.729,Z 858.596,A -85,B 0,C 180,E1 17594.915,E2 17594.915} C_VEL
LIN {X 0,Y 232.21,Z 831.81,A -85,B 0,C 180,E1 17598.333,E2 17598.333} C_VEL
LIN {X 0,Y 232.671,Z 831.81,A -85,B 0,C 180,E1 17611.705,E2 17611.705} C_VEL
LIN {X 0,Y 233.883,Z 831.81,A -85,B 0,C 180,E1 17626.869,E2 17626.869} C_VEL
LIN {X 0,Y 234.926,Z 831.81,A -85,B 0,C 180,E1 17639.859,E2 17639.859} C_VEL
LIN {X 0,Y 234.266,Z 831.81,A -85,B 0,C 180,E1 17648.154,E2 17648.154} C_VEL
LIN {X 0,Y 225.457,Z 831.81,A -85,B 0,C 180,E1 17656.796,E2 17656.796} C_VEL
LIN {X 0,Y 224.392,Z 831.81,A -85,B 0,C 180,E1 17670.476,E2 17670.476} C_VEL
LIN {X 0,Y 224.025,Z 831.81,A -85,B 0,C 180,E1 17685.336,E2 17685.336} C_VEL
LIN {X 0,Y 224.291,Z 831.81,A -85,B 0,C 180,E1 17699.505,E2 17699.505} C_VEL
LIN {X 0,Y 225.314,Z 833.564,A -85,B 0,C 180,E1 17711.773,E2 17711.773} C_VEL
LIN {X 0,Y 242.678,Z 874.654,A -85,B 0,C 180,E1 17717.678,E2 17717.678} C_VEL
LIN {X 0,Y 247.001,Z 907.862,A -85,B 0,C 180,E1 17723.182,E2 17723.182} C_VEL
LIN {X 0,Y 238.188,Z 941.902,A -85,B 0,C 180,E1 17730.912,E2 17730.912} C_VEL
LIN {X 0,Y 232.382,Z 963.073,A -85,B 0,C 180,E1 17740.636,E2 17740.636} C_VEL
LIN {X 0,Y 230.913,Z 971.66,A -85,B 0,C 180,E1 17751.189,E2 17751.189} C_VEL
LIN {X 0,Y 235.847,Z 966.977,A -85,B 0,C 180,E1 17763.156,E2 17763.156} C_VEL
LIN {X 0,Y 246.866,Z 947.552,A -85,B 0,C 180,E1 17773.51,E2 17773.51} C_VEL
LIN {X 0,Y 259.179,Z 916.563,A -85,B 0,C 180,E1 17781.14,E2 17781.14} C_VEL
LIN {X 0,Y 254.154,Z 884.883,A -85,B 0,C 180,E1 17788.905,E2 17788.905} C_VEL
LIN {X 0,Y 238.849,Z 852.44,A -85,B 0,C 180,E1 17798.653,E2 17798.653} C_VEL
LIN {X 0,Y 225.79,Z 831.81,A -85,B 0,C 180,E1 17808.901,E2 17808.901} C_VEL
LIN {X 0,Y 226.913,Z 831.81,A -85,B 0,C 180,E1 17821.92,E2 17821.92} C_VEL
LIN {X 0,Y 225.787,Z 831.81,A -85,B 0,C 180,E1 17833.61,E2 17833.61} C_VEL
LIN {X 0,Y 225.35,Z 833.926,A -85,B 0,C 180,E1 17841.44,E2 17841.44} C_VEL
LIN {X 0,Y 240.95,Z 855.903,A -85,B 0,C 180,E1 17851.831,E2 17851.831} C_VEL
LIN {X 0,Y 260.343,Z 890.6,A -85,B 0,C 180,E1 17860.709,E2 17860.709} C_VEL
LIN {X 0,Y 268.22,Z 921.772,A -85,B 0,C 180,E1 17865.981,E2 17865.981} C_VEL
LIN {X 0,Y 253.461,Z 968.13,A -85,B 0,C 180,E1 17871.598,E2 17871.598} C_VEL
LIN {X 0,Y 238.764,Z 1004.614,A -85,B 0,C 180,E1 17880.491,E2 17880.491} C_VEL
LIN {X 0,Y 229.949,Z 1029.88,A -85,B 0,C 180,E1 17892.725,E2 17892.725} C_VEL
LIN {X 0,Y 229.512,Z 1040.002,A -85,B 0,C 180,E1 17904.309,E2 17904.309} C_VEL
LIN {X 0,Y 229.757,Z 1039.231,A -85,B 0,C 180,E1 17913.788,E2 17913.788} C_VEL
LIN {X 0,Y 229.777,Z 1026.292,A -85,B 0,C 180,E1 17925.293,E2 17925.293} C_VEL
LIN {X 0,Y 235.647,Z 998.013,A -85,B 0,C 180,E1 17936.795,E2 17936.795} C_VEL
LIN {X 0,Y 246.094,Z 958.223,A -85,B 0,C 180,E1 17945.318,E2 17945.318} C_VEL
LIN {X 0,Y 254.68,Z 911.161,A -85,B 0,C 180,E1 17950.551,E2 17950.551} C_VEL
LIN {X 0,Y 237.584,Z 860.268,A -85,B 0,C 180,E1 17955.994,E2 17955.994} C_VEL
LIN {X 0,Y 224.108,Z 831.81,A -85,B 0,C 180,E1 17959.955,E2 17959.955} C_VEL
LIN {X 0,Y 224.756,Z 831.81,A -85,B 0,C 180,E1 17975.717,E2 17975.717} C_VEL
LIN {X 0,Y 226.156,Z 831.81,A -85,B 0,C 180,E1 17990.338,E2 17990.338} C_VEL
LIN {X 0,Y 227.136,Z 831.81,A -85,B 0,C 180,E1 18001.911,E2 18001.911} C_VEL
LIN {X 0,Y 225.457,Z 831.81,A -85,B 0,C 180,E1 18016.796,E2 18016.796} C_VEL
LIN {X 0,Y 216.523,Z 831.81,A -85,B 0,C 180,E1 18025.78,E2 18025.78} C_VEL
LIN {X 0,Y 215.865,Z 831.81,A -85,B 0,C 180,E1 18041.899,E2 18041.899} C_VEL
LIN {X 0,Y 216.199,Z 831.81,A -85,B 0,C 180,E1 18058.234,E2 18058.234} C_VEL
LIN {X 0,Y 217.178,Z 833.585,A -85,B 0,C 180,E1 18070.136,E2 18070.136} C_VEL
LIN {X 0,Y 235.027,Z 874.668,A -85,B 0,C 180,E1 18076.469,E2 18076.469} C_VEL
LIN {X 0,Y 239.736,Z 908.285,A -85,B 0,C 180,E1 18082.269,E2 18082.269} C_VEL
LIN {X 0,Y 230.518,Z 943.274,A -85,B 0,C 180,E1 18090.471,E2 18090.471} C_VEL
LIN {X 0,Y 224.26,Z 965.137,A -85,B 0,C 180,E1 18101.131,E2 18101.131} C_VEL
LIN {X 0,Y 223.415,Z 973.136,A -85,B 0,C 180,E1 18113.513,E2 18113.513} C_VEL
LIN {X 0,Y 229.606,Z 966.512,A -85,B 0,C 180,E1 18125.331,E2 18125.331} C_VEL
LIN {X 0,Y 241.789,Z 945.56,A -85,B 0,C 180,E1 18135.586,E2 18135.586} C_VEL
LIN {X 0,Y 252.678,Z 918.356,A -85,B 0,C 180,E1 18142.24,E2 18142.24} C_VEL
LIN {X 0,Y 248.042,Z 887.167,A -85,B 0,C 180,E1 18150.399,E2 18150.399} C_VEL
LIN {X 0,Y 234.526,Z 857.671,A -85,B 0,C 180,E1 18160.147,E2 18160.147} C_VEL
LIN {X 0,Y 221.948,Z 838.707,A -85,B 0,C 180,E1 18170.41,E2 18170.41} C_VEL
LIN {X 0,Y 218.637,Z 831.81,A -85,B 0,C 180,E1 18176.024,E2 18176.024} C_VEL
LIN {X 0,Y 218.549,Z 831.81,A -85,B 0,C 180,E1 18185.983,E2 18185.983} C_VEL
LIN {X 0,Y 218.044,Z 834.012,A -85,B 0,C 180,E1 18193.833,E2 18193.833} C_VEL
LIN {X 0,Y 224.542,Z 843.771,A -85,B 0,C 180,E1 18201.827,E2 18201.827} C_VEL
LIN {X 0,Y 238.659,Z 863.467,A -85,B 0,C 180,E1 18211.322,E2 18211.322} C_VEL
LIN {X 0,Y 256.165,Z 897.574,A -85,B 0,C 180,E1 18220.285,E2 18220.285} C_VEL
LIN {X 0,Y 261.631,Z 924.834,A -85,B 0,C 180,E1 18225.033,E2 18225.033} C_VEL
LIN {X 0,Y 246.252,Z 969.732,A -85,B 0,C 180,E1 18230.828,E2 18230.828} C_VEL
LIN {X 0,Y 230.495,Z 1006.28,A -85,B 0,C 180,E1 18240.411,E2 18240.411} C_VEL
LIN {X 0,Y 221.817,Z 1030.105,A -85,B 0,C 180,E1 18253.076,E2 18253.076} C_VEL
LIN {X 0,Y 221.553,Z 1038.83,A -85,B 0,C 180,E1 18264.104,E2 18264.104} C_VEL
LIN {X 0,Y 221.846,Z 1037.928,A -85,B 0,C 180,E1 18273.923,E2 18273.923} C_VEL
LIN {X 0,Y 222.229,Z 1023.179,A -85,B 0,C 180,E1 18286.763,E2 18286.763} C_VEL
LIN {X 0,Y 228.791,Z 994.33,A -85,B 0,C 180,E1 18298.203,E2 18298.203} C_VEL
LIN {X 0,Y 239.752,Z 953.754,A -85,B 0,C 180,E1 18306.682,E2 18306.682} C_VEL
LIN {X 0,Y 247.313,Z 912.081,A -85,B 0,C 180,E1 18311.378,E2 18311.378} C_VEL
LIN {X 0,Y 230.994,Z 862.741,A -85,B 0,C 180,E1 18317.023,E2 18317.023} C_VEL
LIN {X 0,Y 216.094,Z 831.81,A -85,B 0,C 180,E1 18321.473,E2 18321.473} C_VEL
LIN {X 0,Y 216.833,Z 831.81,A -85,B 0,C 180,E1 18337.355,E2 18337.355} C_VEL
LIN {X 0,Y 218.099,Z 831.81,A -85,B 0,C 180,E1 18349.978,E2 18349.978} C_VEL
LIN {X 0,Y 219.099,Z 831.81,A -85,B 0,C 180,E1 18361.981,E2 18361.981} C_VEL
LIN {X 0,Y 217.327,Z 831.81,A -85,B 0,C 180,E1 18376.762,E2 18376.762} C_VEL
LIN {X 0,Y 216.523,Z 831.81,A -85,B 0,C 180,E1 18385.78,E2 18385.78} C_VEL
LIN {X 0,Y 207.773,Z 831.81,A -85,B 0,C 180,E1 18395.093,E2 18395.093} C_VEL
LIN {X 0,Y 207.73,Z 831.81,A -85,B 0,C 180,E1 18410.088,E2 18410.088} C_VEL
LIN {X 0,Y 208.421,Z 831.81,A -85,B 0,C 180,E1 18425.522,E2 18425.522} C_VEL
LIN {X 0,Y 209.04,Z 833.933,A -85,B 0,C 180,E1 18428.364,E2 18428.364} C_VEL
